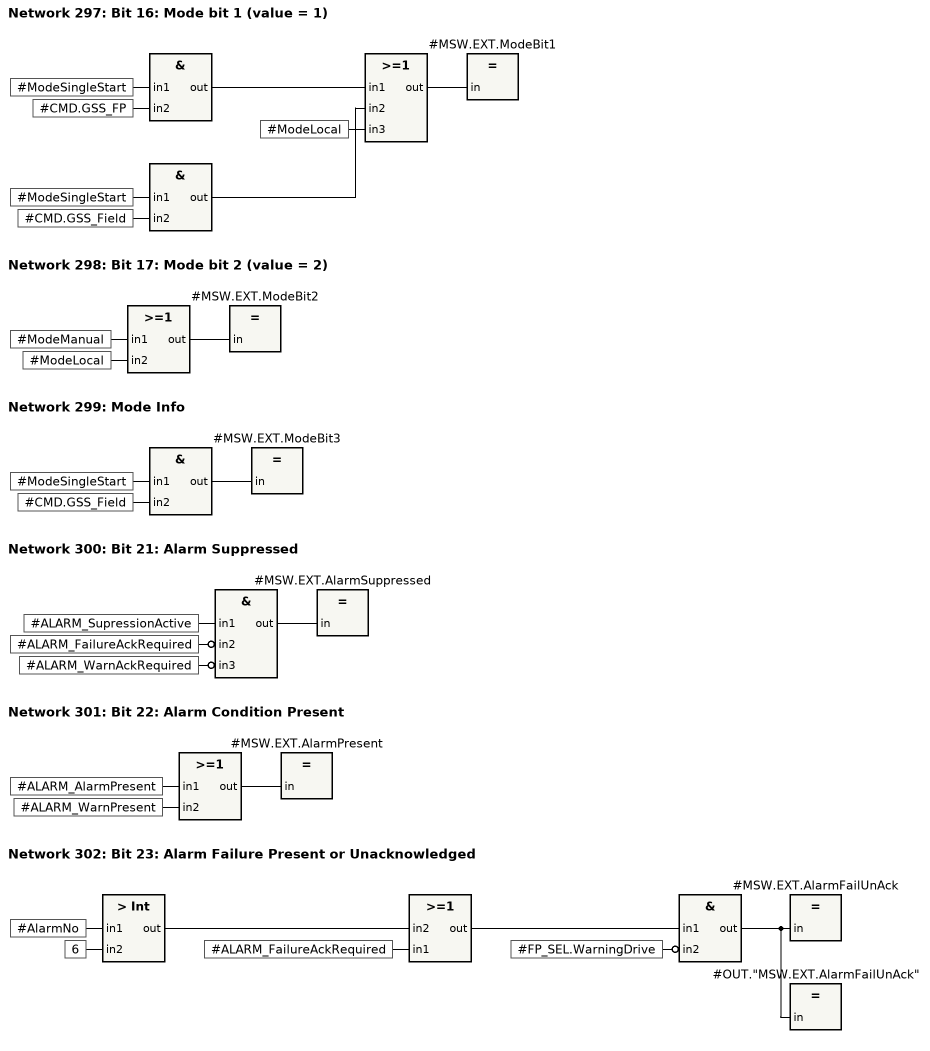
   #MSW.EXT.ModeBit1 := (#ModeSingleStart AND #CMD.GSS_FP) OR (#ModeSingleStart AND #CMD.GSS_Field) OR #ModeLocal;
END_REGION

REGION Network 298: Bit 17: Mode bit 2 (value = 2)
   #MSW.EXT.ModeBit2 := #ModeManual OR #ModeLocal;
END_REGION

REGION Network 299: Mode Info
   #MSW.EXT.ModeBit3 := #ModeSingleStart AND #CMD.GSS_Field;
END_REGION

REGION Network 300: Bit 21: Alarm Suppressed
   #MSW.EXT.AlarmSuppressed := #ALARM_SupressionActive AND NOT #ALARM_FailureAckRequired AND NOT #ALARM_WarnAckRequired;
END_REGION

REGION Network 301: Bit 22: Alarm Condition Present
   #MSW.EXT.AlarmPresent := #ALARM_AlarmPresent OR #ALARM_WarnPresent;
END_REGION

REGION Network 302: Bit 23: Alarm Failure Present or Unacknowledged
   #MSW.EXT.AlarmFailUnAck := ((#AlarmNo > 6) OR #ALARM_FailureAckRequired) AND NOT #FP_SEL.WarningDrive;
   #OUT."MSW.EXT.AlarmFailUnAck" := #MSW.EXT.AlarmFailUnAck;
END_REGION

REGION Network 303: Bit 24: Alarm Warning Present or Unacknowledged
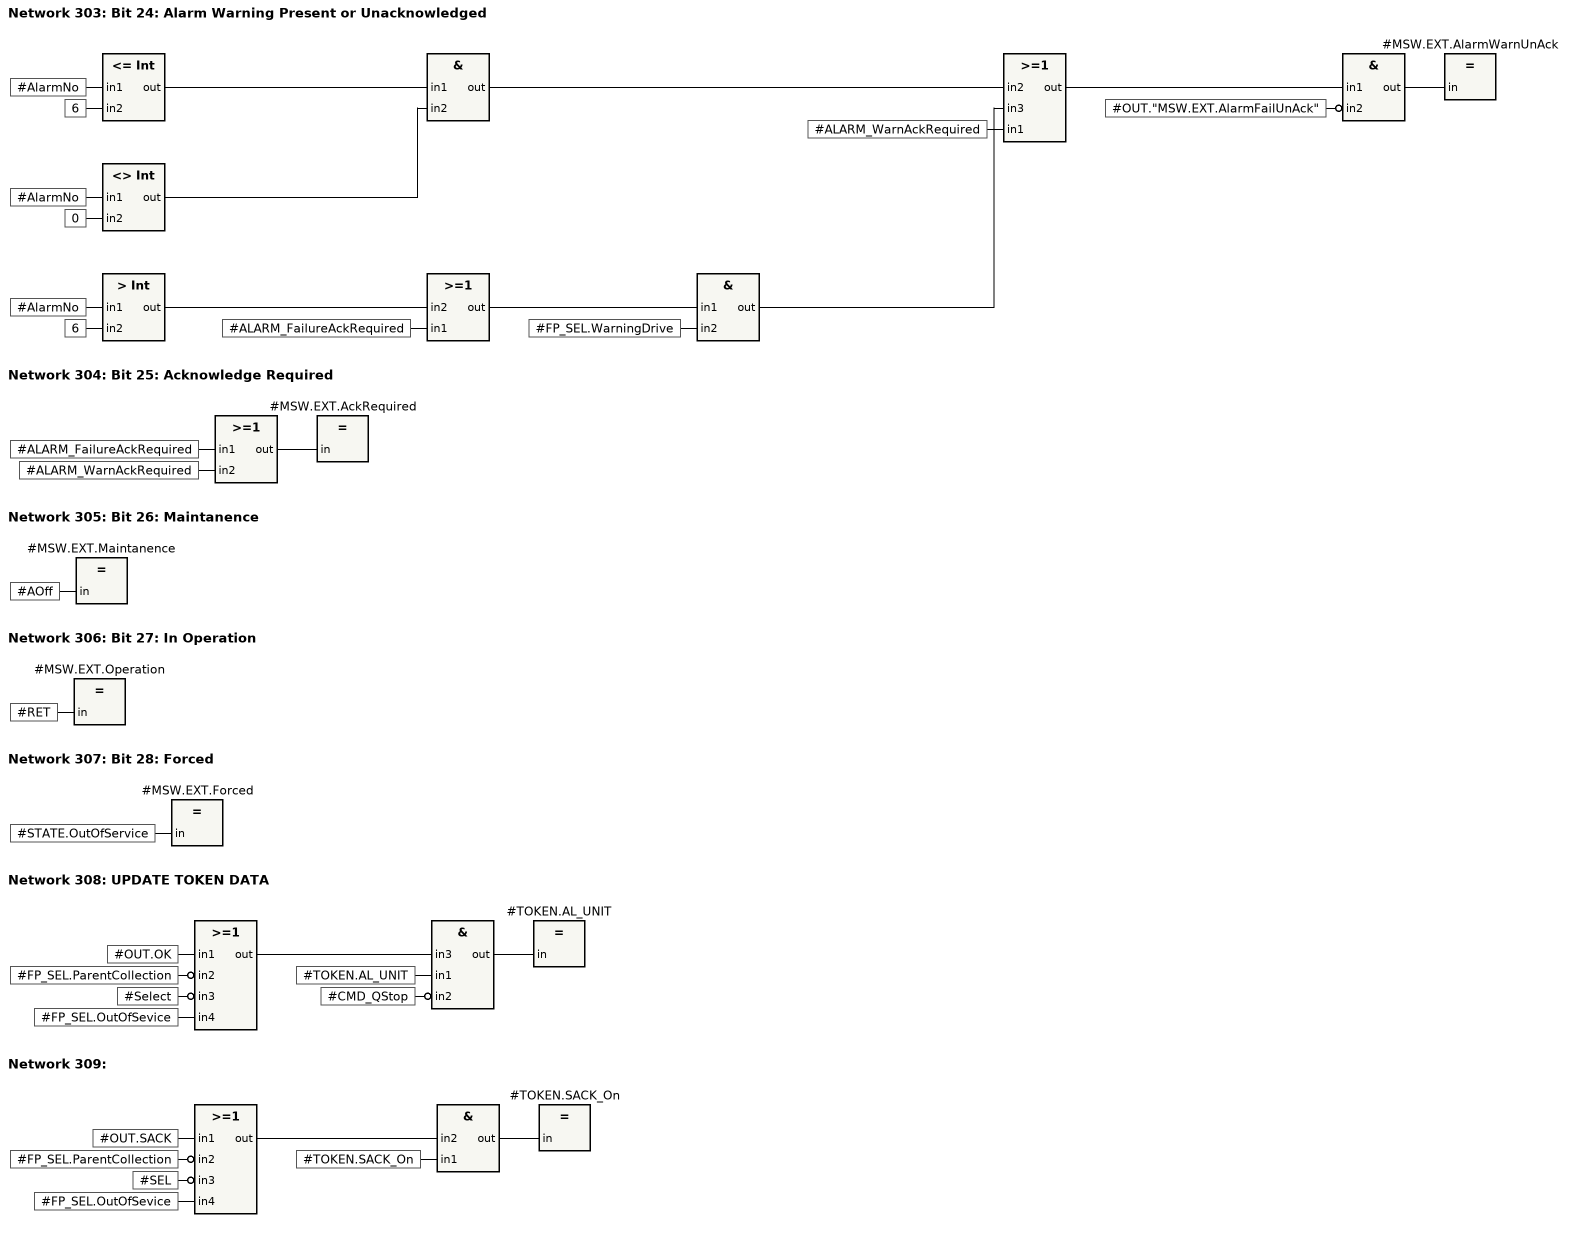
   #MSW.EXT.AlarmWarnUnAck := (((#AlarmNo <= 6) AND (#AlarmNo <> 0)) OR (((#AlarmNo > 6) OR #ALARM_FailureAckRequired) AND #FP_SEL.WarningDrive) OR #ALARM_WarnAckRequired) AND NOT #OUT."MSW.EXT.AlarmFailUnAck";
END_REGION

REGION Network 304: Bit 25: Acknowledge Required
   #MSW.EXT.AckRequired := #ALARM_FailureAckRequired OR #ALARM_WarnAckRequired;
END_REGION

REGION Network 305: Bit 26: Maintanence
   #MSW.EXT.Maintanence := #AOff;
END_REGION

REGION Network 306: Bit 27: In Operation
   #MSW.EXT.Operation := #RET;
END_REGION

REGION Network 307: Bit 28: Forced
   // Build 002 - 27 March 2018: OuOfService condition would show Force icon (bit 28)
   #MSW.EXT.Forced := #STATE.OutOfService;
END_REGION

REGION Network 308: UPDATE TOKEN DATA
   #TOKEN.AL_UNIT := (#OUT.OK OR NOT #FP_SEL.ParentCollection OR NOT #Select OR #FP_SEL.OutOfSevice) AND #TOKEN.AL_UNIT AND NOT #CMD_QStop;
END_REGION

REGION Network 309
   // Build 005 - 24.Jun.2020 (MIA-US): Replace "Select" with "SEL"
   #TOKEN.SACK_On := (#OUT.SACK OR NOT #FP_SEL.ParentCollection OR NOT #SEL OR #FP_SEL.OutOfSevice) AND #TOKEN.SACK_On;
END_REGION

REGION Network 310
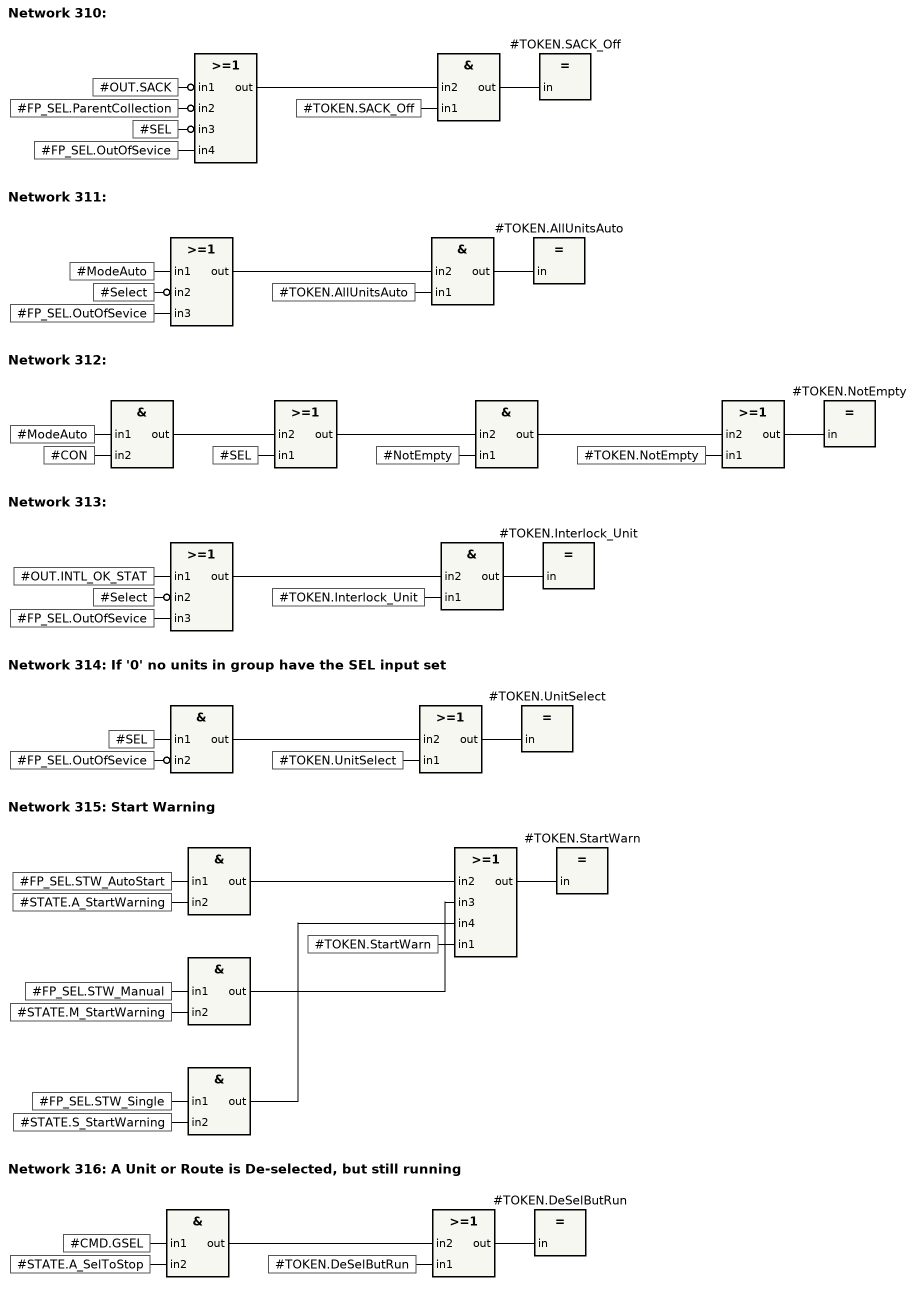
   #TOKEN.SACK_Off := (NOT #OUT.SACK OR NOT #FP_SEL.ParentCollection OR NOT #SEL OR #FP_SEL.OutOfSevice) AND #TOKEN.SACK_Off;
END_REGION

REGION Network 311
   #TOKEN.AllUnitsAuto := (#ModeAuto OR NOT #Select OR #FP_SEL.OutOfSevice) AND #TOKEN.AllUnitsAuto;
END_REGION

REGION Network 312
   #TOKEN.NotEmpty := (((#ModeAuto AND #CON) OR #SEL) AND #NotEmpty) OR #TOKEN.NotEmpty;
END_REGION

REGION Network 313
   #TOKEN.Interlock_Unit := (#OUT.INTL_OK_STAT OR NOT #Select OR #FP_SEL.OutOfSevice) AND #TOKEN.Interlock_Unit;
END_REGION

REGION Network 314: If '0' no units in group have the SEL input set
   #TOKEN.UnitSelect := (#SEL AND NOT #FP_SEL.OutOfSevice) OR #TOKEN.UnitSelect;
END_REGION

REGION Network 315: Start Warning
   #TOKEN.StartWarn := (#FP_SEL.STW_AutoStart AND #STATE.A_StartWarning) OR (#FP_SEL.STW_Manual AND #STATE.M_StartWarning) OR (#FP_SEL.STW_Single AND #STATE.S_StartWarning) OR #TOKEN.StartWarn;
END_REGION

REGION Network 316: A Unit or Route is De-selected, but still running
   #TOKEN.DeSelButRun := (#CMD.GSEL AND #STATE.A_SelToStop) OR #TOKEN.DeSelButRun;
END_REGION

REGION Network 317: Interlock
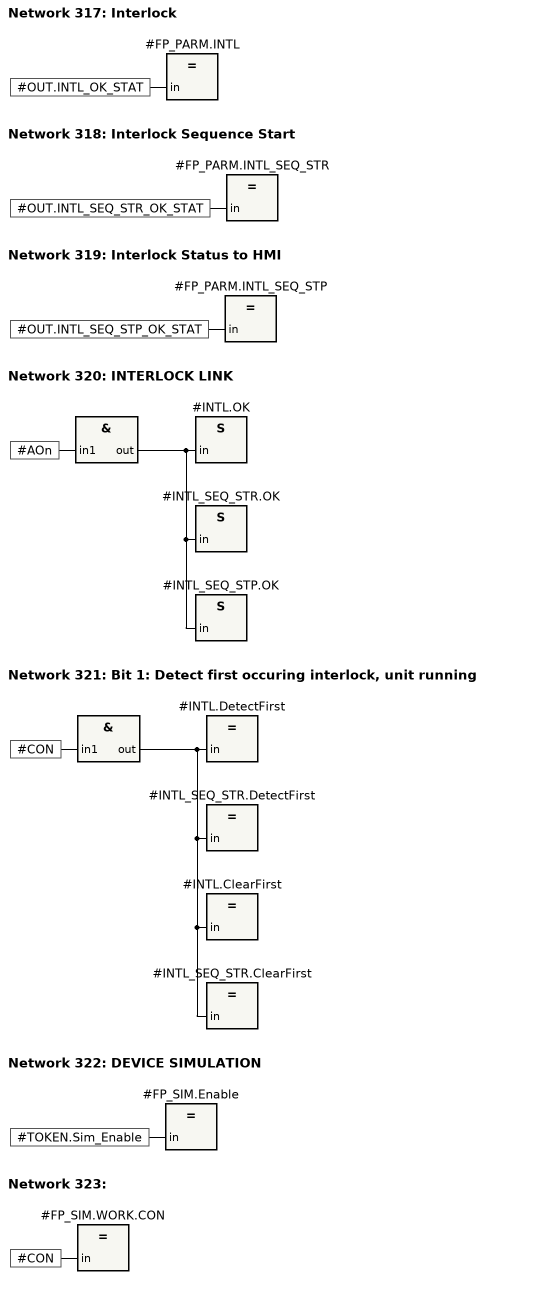
   #FP_PARM.INTL := #OUT.INTL_OK_STAT;
END_REGION

REGION Network 318: Interlock Sequence Start
   #FP_PARM.INTL_SEQ_STR := #OUT.INTL_SEQ_STR_OK_STAT;
END_REGION

REGION Network 319: Interlock Status to HMI
   #FP_PARM.INTL_SEQ_STP := #OUT.INTL_SEQ_STP_OK_STAT;
END_REGION

REGION Network 320: INTERLOCK LINK
   IF #AOn THEN
       #INTL.OK := TRUE;
       #INTL_SEQ_STR.OK := TRUE;
       #INTL_SEQ_STP.OK := TRUE;
   END_IF;
END_REGION

REGION Network 321: Bit 1: Detect first occuring interlock, unit running
   #INTL.DetectFirst := #CON;
   #INTL_SEQ_STR.DetectFirst := #CON;
   #INTL.ClearFirst := #CON;
   #INTL_SEQ_STR.ClearFirst := #CON;
END_REGION

REGION Network 322: DEVICE SIMULATION
   #FP_SIM.Enable := #TOKEN.Sim_Enable;
END_REGION

REGION Network 323
   #FP_SIM.WORK.CON := #CON;
END_REGION

REGION Network 324
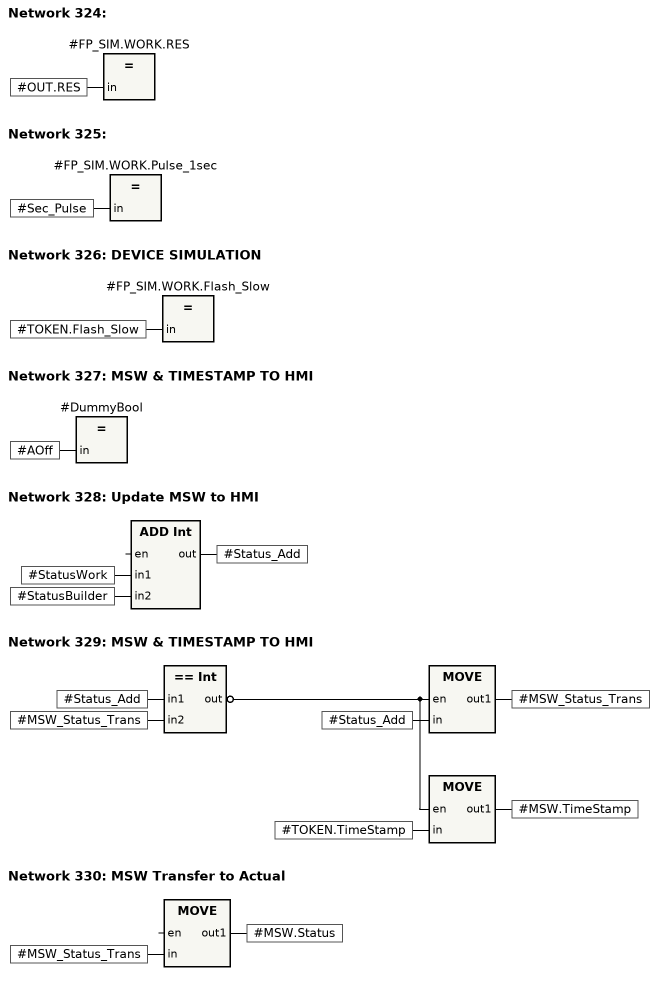
   #FP_SIM.WORK.RES := #OUT.RES;
END_REGION

REGION Network 325
   #FP_SIM.WORK.Pulse_1sec := #Sec_Pulse;
END_REGION

REGION Network 326: DEVICE SIMULATION
   #FP_SIM.WORK.Flash_Slow := #TOKEN.Flash_Slow;
END_REGION

REGION Network 327: MSW & TIMESTAMP TO HMI
   Done:
   #DummyBool := #AOff;
END_REGION

REGION Network 328: Update MSW to HMI
   #Status_Add := #StatusWork + #StatusBuilder;
END_REGION

REGION Network 329: MSW & TIMESTAMP TO HMI
   #_w1 := NOT (#Status_Add = #MSW_Status_Trans);
   IF #_w1 THEN
       #MSW_Status_Trans := #Status_Add;
       #MSW.TimeStamp := #TOKEN.TimeStamp;
   END_IF;
END_REGION

REGION Network 330: MSW Transfer to Actual
   #MSW.Status := #MSW_Status_Trans;
END_REGION

REGION Network 331: Write STAT to OUT
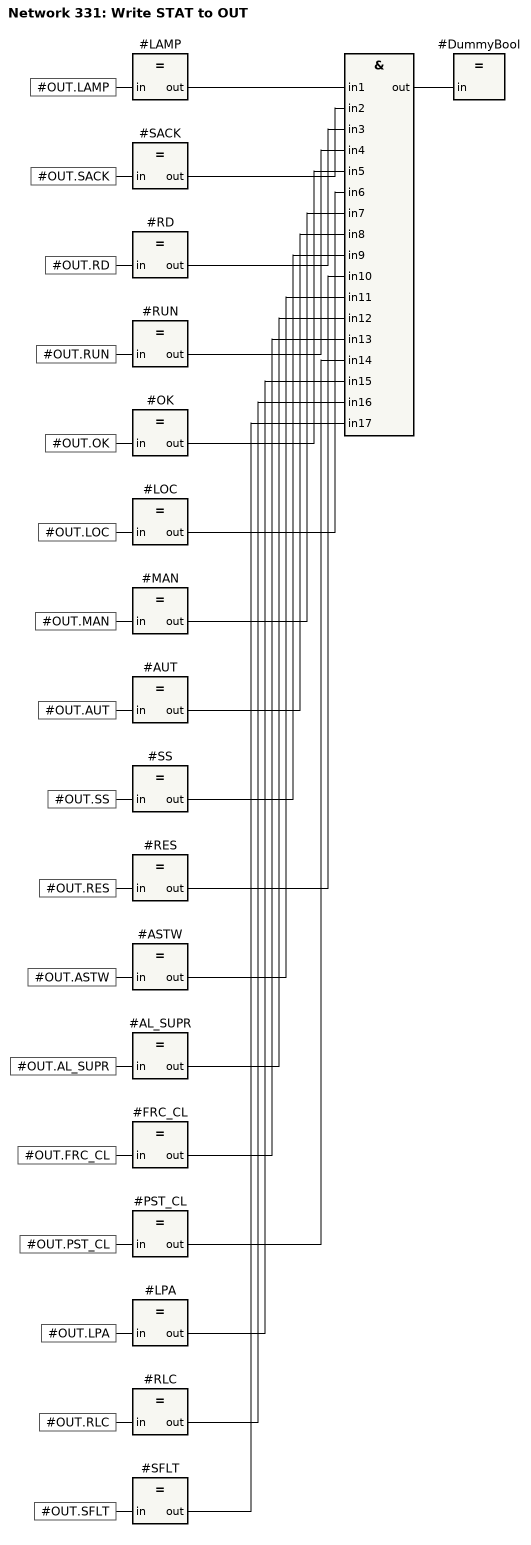
   #LAMP := #OUT.LAMP;
   #SACK := #OUT.SACK;
   #RD := #OUT.RD;
   #RUN := #OUT.RUN;
   #OK := #OUT.OK;
   #LOC := #OUT.LOC;
   #MAN := #OUT.MAN;
   #AUT := #OUT.AUT;
   #SS := #OUT.SS;
   #RES := #OUT.RES;
   #ASTW := #OUT.ASTW;
   #AL_SUPR := #OUT.AL_SUPR;
   #FRC_CL := #OUT.FRC_CL;
   #PST_CL := #OUT.PST_CL;
   #LPA := #OUT.LPA;
   #RLC := #OUT.RLC;
   #SFLT := #OUT.SFLT;
   #DummyBool := #OUT.LAMP AND #OUT.SACK AND #OUT.RD AND #OUT.RUN AND #OUT.OK AND #OUT.LOC AND #OUT.MAN AND #OUT.AUT AND #OUT.SS AND #OUT.RES AND #OUT.ASTW AND #OUT.AL_SUPR AND #OUT.FRC_CL AND #OUT.PST_CL AND #OUT.LPA AND #OUT.RLC AND #OUT.SFLT;
END_REGION
END_FUNCTION_BLOCK

FUNCTION_BLOCK "ACESYS_PFISTER_SDD"   // FB218, SCL
TITLE = ACESYS V8.0 - Build 005 - PFISTER SDD Block
{ S7_Optimized_Access := 'FALSE' }
AUTHOR : FLSmidth
FAMILY : ACESYS
NAME : PFISTER_SDD
VERSION : 8.0
   VAR_INPUT
      CMD : "ACESYS_GRP_CMD";
      SEL : Bool;
      ASTR : Bool;
      SSW : Bool;
      DOS_SP : Real;
      MEAS_SP : Real;
      OPT_VAL_RATIO : Int;
   END_VAR
   VAR_OUTPUT
      INTL : "ACESYS_INTL";
      INTL_SEQ_STR : "ACESYS_INTL";
      INTL_SEQ_STP : "ACESYS_INTL";
      LAMP : Bool;
      SACK : Bool;
      RD : Bool;
      RUN : Bool;
      OK : Bool;
      WARN : Bool;
      LOC : Bool;
      MAN : Bool;
      AUT : Bool;
      SS : Bool;
      ASTW : Bool;
      AL_SUPR : Bool;
      DOS : Bool;
      MEAS : Bool;
      FEED_Pct : Real;
      FEED_Eng : Real;
      SPEED_Pct : Real;
      SPEED_Eng : Real;
      LOAD_Pct : Real;
      TOT_Pulse : Bool;
      ERROR_CODE : Int;
      MSW : "ACESYS_HMI_STAT_32T";
   END_VAR
   VAR_IN_OUT
      TOKEN : "ACESYS_TOKEN";
   END_VAR
   VAR
      BlockInfo : Struct
         Ace_Version : Int;
         Ace_BuildNo : Int;
         State_Act : Int;
         State_Prev : Int;
         DB_Number : Int;
      END_STRUCT;
      FP_CMD : Struct
         QuickStop : Bool;
         SetUserCorr : Bool;
         Auto : Bool;
         Manual : Bool;
         Local : Bool;
         Start : Bool;
         Reset : Bool;
         AckAlarm : Bool;
         Stop : Bool;
         Measuring : Bool;
         Dosing : Bool;
         Spare_04 : Bool;
         Spare_03 : Bool;
         Spare_02 : Bool;
         Spare_01 : Bool;
         Spare_00 : Bool;
      END_STRUCT;
      FP_SEL : Struct
         STW_AutoStart : Bool;
         STW_Manual : Bool;
         STW_Single : Bool;
         STW_Local : Bool;
         ParentSupress : Bool;
         ParentCollection : Bool;
         OutOfSevice : Bool;
         Spare_00 : Bool;
         Spare_01 : Bool;
         Spare_02 : Bool;
         Spare_03 : Bool;
         Spare_04 : Bool;
         Spare_05 : Bool;
         Spare_06 : Bool;
         Spare_07 : Bool;
         Spare_08 : Bool;
      END_STRUCT;
      FP_EN : Struct
         Mode_Auto : Bool;
         Mode_Man : Bool;
         Mode_Loc : Bool;
         Mode_SS_Field : Bool;
         Mode_SS_FP : Bool;
         PB_QStop : Bool;
         Spare_00 : Bool;
         Spare_01 : Bool;
         Spare_02 : Bool;
         Spare_03 : Bool;
         Spare_04 : Bool;
         Spare_05 : Bool;
         Spare_06 : Bool;
         Spare_07 : Bool;
         Spare_08 : Bool;
         Spare_09 : Bool;
      END_STRUCT;
      FP_DIM : Struct
         Auto : Bool;
         Local : Bool;
         Manual : Bool;
         Start : Bool;
         Stop : Bool;
         QStop : Bool;
         Measuring : Bool;
         Dosing : Bool;
         Reset : Bool;
         SetUserCorr : Bool;
         Spare6 : Bool;
         Spare5 : Bool;
         Spare4 : Bool;
         Spare3 : Bool;
         Spare2 : Bool;
         Spare1 : Bool;
      END_STRUCT;
      FP_SHOW : Struct
         PB_Auto : Bool;
         PB_Local : Bool;
         PB_Manual : Bool;
         PB_Start : Bool;
         PB_Stop : Bool;
         PB_QStop : Bool;
         ACK : Bool;
         PB_Dosing : Bool;
         PB_Measuring : Bool;
         PB_Reset : Bool;
         Feedrate : Bool;
         Load : Bool;
         Speed : Bool;
         Preload : Bool;
         Current : Bool;
         Droppointload : Bool;
      END_STRUCT;
      FP_PARM : Struct
         INTL : Bool;
         INTL_SEQ_STR : Bool;
         INTL_SEQ_STP : Bool;
         CorrAccepted : Bool;
         SelectVal_Enable : Bool;
         Run : Bool;
         Spare02 : Bool;
         Spare01 : Bool;
         StartWarn_Pre : DInt;
         StartWarn_Acc : DInt;
         RunDelay_Pre : DInt;
         RunDelay_Acc : DInt;
         DelayStart_Pre : DInt;
         DelayStart_Acc : DInt;
         DelayStop_Pre : DInt;
         DelayStop_Acc : DInt;
         ReturnMon_Pre : DInt;
         ReturnMon_Acc : DInt;
         CORR_User : Real;
         Measuring_SP : Real;
         Dosing_SP : Real;
         Feedrate_SP : Real;
         Act_Feedrate : Int;
         Act_Load : Int;
         Act_Speed : Int;
         Act_Preload : Int;
         Act_Current : Int;
         Act_Droppointload : Int;
         OptValRatio : Int;
         StopReason : Int;
         PresentError : Int;
         LastError : Int;
         PresentWarning : Int;
         LastWarning : Int;
         Range_Feed : Real;
         Range_Speed : Real;
      END_STRUCT;
      FP_SIM : "ACESYS_SIM_PFISTER_SDD";
      AdapterBlock : "ACESYS_ADPT_PFISTERSDD";
      STATE : Struct
         A_AutoStart : Bool;
         A_DelayedStart : Bool;
         A_DelayedStop : Bool;
         A_Running : Bool;
         A_Selected : Bool;
         A_SelToStop : Bool;
         A_Stopping : Bool;
         A_SeqStart : Bool;
         A_SeqStop : Bool;
         A_Starting : Bool;
         A_StartWarning : Bool;
         A_Stopped : Bool;
         A_EmptyingSystem : Bool;
         S_AutoStart : Bool;
         S_Running : Bool;
         S_Starting : Bool;
         S_StartWarning : Bool;
         S_Stopped : Bool;
         S_Stopping : Bool;
         S_EmptyingSystem : Bool;
         M_Running : Bool;
         M_Starting : Bool;
         M_StartWarning : Bool;
         M_Stopped : Bool;
         M_Stopping : Bool;
         M_EmptyingSystem : Bool;
         L_Running : Bool;
         L_Stopped : Bool;
         Alarm : Bool;
         Interlock : Bool;
         EmergencyStop : Bool;
         OutOfService : Bool;
      END_STRUCT;
      ONS : Struct
         AckAlarm : Bool;
         Cmd_Auto : Bool;
         Cmd_Manual : Bool;
         Cmd_Local : Bool;
         Cmd_Start : Bool;
         Cmd_Measuring : Bool;
         Cmd_Dosing : Bool;
         GLTP : Bool;
         FP_Start_CMD : Bool;
         SetUserCorr : Bool;
         ResetTot : Bool;
         Reset : Bool;
         Sec_Pulse1 : Bool;
         Sec_Pulse2 : Bool;
      END_STRUCT;
      Pulse_Flag : Struct
         AckAlarm : Bool;
         Cmd_Auto : Bool;
         Cmd_Manual : Bool;
         Cmd_Local : Bool;
         Cmd_Start : Bool;
         Cmd_Measuring : Bool;
         Cmd_Dosing : Bool;
         GLTP : Bool;
         FP_Start_CMD : Bool;
         SetUserCorr : Bool;
         ResetTot : Bool;
         Reset : Bool;
         Sec_Pulse1 : Bool;
         Sec_Pulse2 : Bool;
      END_STRUCT;
      StatusWork : Int;
      AlarmNo : Int;
      AlarmNo_Old : Int;
      RET_VAL_Output : Int;
      RET_VAL_Input : Int;
      SelectVal_Count : Int;
      ModePointer : Int;
      DelayStart_Pre : DInt;
      DelayStart_Acc : DInt;
      DelayStop_Pre : DInt;
      DelayStop_Acc : DInt;
      StartWarn_Pre : DInt;
      StartWarn_Acc : DInt;
      RunDelay_Pre : DInt;
      RunDelay_Acc : DInt;
      ReturnMon_Pre : DInt;
      ReturnMon_Acc : DInt;
      DelayStart_Mem : DInt;
      DelayStop_Mem : DInt;
      StartWarn_Mem : DInt;
      RunDelay_Mem : DInt;
      ReturnMon_Mem : DInt;
      GWA : Bool;
      GFA : Bool;
      CMD_AckAlarm : Bool;
      CMD_Start : Bool;
      CMD_Stop : Bool;
      CMD_QStop : Bool;
      CMD_Measuring : Bool;
      CMD_Dosing : Bool;
      FromStateAuto : Bool;
      FromStateSingle : Bool;
      FromStateManual : Bool;
      FromStateLocal : Bool;
      FromStopState : Bool;
      ALARM_SupressionActive : Bool;
      ALARM_AlarmPresent : Bool;
      ALARM_WarnPresent : Bool;
      ALARM_FailureAckRequired : Bool;
      ALARM_WarnAckRequired : Bool;
      StartWarn_TT : Bool;
      StartWarn_Done : Bool;
      Rundelay_Done : Bool;
      DelayStart_Done : Bool;
      DelayStop_Done : Bool;
      ReturnMon_Done : Bool;
      Trig_RET_ALARM : Bool;
      RET_OneScan : Bool;
      NotEmpty : Bool;
      Sec_Pulse : Bool;
      Start : Bool;
      ModeAuto : Bool;
      ModeLocal : Bool;
      ModeManual : Bool;
      ModeSingleStart : Bool;
      ModeMeasuring : Bool;
      ModeDosing : Bool;
      Select : Bool;
      BitVar : Bool;
      OUT : Struct
         LAMP : Bool;
         SACK : Bool;
         RD : Bool;
         RUN : Bool;
         OK : Bool;
         WARN : Bool;
         LOC : Bool;
         MAN : Bool;
         AUT : Bool;
         SS : Bool;
         ASTW : Bool;
         AL_SUPR : Bool;
         DOS : Bool;
         MEAS : Bool;
         INTL_OK_STAT : Bool;
         INTL_SEQ_STR_OK_STAT : Bool;
         INTL_SEQ_STP_OK_STAT : Bool;
         ERROR_CODE : Int;
      END_STRUCT;
      DelayStart_Timer : TON_TIME;
      DelayStop_Timer : TON_TIME;
      StartWarn_Timer : TON_TIME;
      RunDelay_Timer : TON_TIME;
      ReturnMon_Timer : TON_TIME;
      UserCorr_Timer : TON_TIME;
      Reset_Timer : TON_TIME;
      WatchDog_Timer : TON_TIME;
   END_VAR
   VAR_TEMP
      AOn : Bool;
      AOff : Bool;
      Temp_CON : Bool;
      BusFault : Bool;
      WatchDog_Elapsed : Bool;
      WatchDog_Same : Bool;
      SelectVal_Same : Bool;
      DummyBool : Bool;
      DummyBool1 : Bool;
      DummyBool2 : Bool;
      DummyBool3 : Bool;
      DummyReal : Real;
      DummyWord : Word;
      DummyDWord : DWord;
      DummyDInt : DInt;
      DummyInt : Int;
      StatPointer_Old : Int;
      StatusBuilder : Int;
      Status_Add : Int;
      Error_Old : Int;
      Warning_Old : Int;
      AnyPtr : ANY;
      AnyStruct AT AnyPtr : Struct
         S7_ID : Byte;
         Mem_ID : Byte;
         NumberOfElements : Int;
         DB_Number : Word;
         BitPointer : DWord;
      END_STRUCT;
   END_VAR
BEGIN
   (* ----------------------------------------------------------------- Block Information -------------------------------------------------------------*)
   (* Version AND Build No *)
   #BlockInfo.Ace_Version := 80;
   #BlockInfo.Ace_BuildNo := 5;

   (* INSTANCE DB Number TO Faceplate *)
   #AnyPtr := #BitVar;
   #BlockInfo.DB_Number := WORD_TO_INT(#AnyStruct.DB_Number);

   (* Second Pulse *)
   #Pulse_Flag.Sec_Pulse1 := #TOKEN.SEC_Toggle AND NOT #ONS.Sec_Pulse1;
   #ONS.Sec_Pulse1 := #TOKEN.SEC_Toggle;

   #Pulse_Flag.Sec_Pulse2 := NOT #TOKEN.SEC_Toggle AND NOT #ONS.Sec_Pulse2;
   #ONS.Sec_Pulse2 := NOT #TOKEN.SEC_Toggle;

   #Sec_Pulse := #Pulse_Flag.Sec_Pulse1 OR #Pulse_Flag.Sec_Pulse2;
   #Pulse_Flag.ResetTot := #Sec_Pulse OR #Pulse_Flag.ResetTot;

   #OUT.INTL_OK_STAT := PEEK_BOOL(area := 16#84, dbNumber := #BlockInfo.DB_Number, byteOffset := 14, bitOffset := 0);
   #OUT.INTL_SEQ_STR_OK_STAT := PEEK_BOOL(area := 16#84, dbNumber := #BlockInfo.DB_Number, byteOffset := 16, bitOffset := 0);
   #OUT.INTL_SEQ_STP_OK_STAT := PEEK_BOOL(area := 16#84, dbNumber := #BlockInfo.DB_Number, byteOffset := 18, bitOffset := 0);

   (* ----------------------------------------------------------------- Initialization ------------------------------------------------------------- *)
   (* ---- WatchDog ---- *)

   IF #FP_SIM.Enable THEN
       #WatchDog_Same := #AdapterBlock.Togglebit_T = #FP_SIM.WORK.Togglebit;
   ELSE
       #WatchDog_Same := #AdapterBlock.Togglebit_R = #AdapterBlock.Togglebit_T;
   END_IF;

   #WatchDog_Timer(IN := NOT #WatchDog_Same,
                   PT := INT_TO_DINT(3000),
                   ET => #DummyDInt,
                   Q => #WatchDog_Elapsed);


   IF #FP_SIM.Enable THEN
       #AdapterBlock.Togglebit_T := NOT #FP_SIM.WORK.Togglebit;
   ELSE
       #AdapterBlock.Togglebit_T := NOT #AdapterBlock.Togglebit_R;
   END_IF;
   #BusFault := NOT (#FP_SIM.Enable AND  #WatchDog_Elapsed);

   (* ---- #Select ---- *)
   #Select := #CMD.GSEL AND #SEL;

   (* // ---- Init Modes ---- *)
   IF NOT #FP_EN.Mode_Auto AND NOT #FP_EN.Mode_Loc AND NOT #FP_EN.Mode_Man AND NOT #FP_EN.Mode_SS_Field AND NOT #FP_EN.Mode_SS_FP THEN
       #FP_EN.Mode_Auto := TRUE;
       #FP_EN.Mode_Man := TRUE;
       #FP_EN.Mode_Loc := TRUE;
       #FP_EN.Mode_SS_FP := TRUE;
   END_IF;

   IF NOT #CMD_Measuring AND NOT #CMD_Dosing THEN
       #CMD_Measuring := TRUE;
   END_IF;

   (* // ---- Show Push Buttons ---- *)
   #FP_SHOW.PB_Auto := NOT #FP_SEL.OutOfSevice AND #FP_EN.Mode_Auto;
   #FP_SHOW.PB_Local := NOT #FP_SEL.OutOfSevice AND #FP_EN.Mode_Loc AND #TOKEN.Loc_Enable AND NOT #TOKEN.REM_TYPE;
   #FP_SHOW.PB_Manual := NOT #FP_SEL.OutOfSevice AND #FP_EN.Mode_Man AND #TOKEN.Man_Enable;
   #FP_SHOW.PB_Start := NOT #FP_SEL.OutOfSevice AND (#FP_EN.Mode_Man OR #FP_EN.Mode_SS_FP);
   #FP_SHOW.PB_Stop := NOT #FP_SEL.OutOfSevice AND (#FP_EN.Mode_Man OR #FP_EN.Mode_SS_FP);
   #FP_SHOW.PB_QStop := NOT #FP_SEL.OutOfSevice AND #FP_EN.PB_QStop AND #TOKEN.QSTOP_FP_Unit;

   IF #FP_SIM.Enable THEN
       #FP_PARM.Run := #FP_SIM.WORK.Run;
   ELSE
       #FP_PARM.Run := #AdapterBlock.Run;
   END_IF;



   (* // ----------------------------------------------------------------- FacePlate DimOuts -------------------------------------------------------------//  *)
   (* // ---- DimOut Buttons ---- *)
   (* // Auto Button *)
   #FP_DIM.Auto := #ModeLocal OR #ModeManual;
   #FP_DIM.Auto := #FP_DIM.Auto AND NOT (#TOKEN.LOC_TYPE AND #ModeLocal AND #FP_PARM.Run);
   #FP_DIM.Auto := #FP_DIM.Auto AND NOT (#ModeLocal AND #CMD.GLTP);
   #FP_DIM.Auto := #FP_DIM.Auto AND #FP_SHOW.PB_Auto AND #TOKEN.EmergencyStop;
   (* // Manual Button *)
   #FP_DIM.Manual := #ModeLocal AND NOT #TOKEN.LOC_TYPE;
   #FP_DIM.Manual := #FP_DIM.Manual OR (#ModeLocal AND #TOKEN.LOC_TYPE AND NOT #FP_PARM.Run);
   #FP_DIM.Manual := #FP_DIM.Manual OR (#ModeAuto AND NOT #Select AND NOT #STATE.A_SelToStop AND NOT #STATE.A_Stopping AND NOT #STATE.A_Selected);
   #FP_DIM.Manual := #FP_DIM.Manual AND NOT (#ModeLocal AND #CMD.GLTP);
   #FP_DIM.Manual := #FP_DIM.Manual AND #FP_SHOW.PB_Manual AND #TOKEN.EmergencyStop;
   (* // Local Button *)
   #FP_DIM.Local := #ModeAuto AND NOT #Select AND NOT #STATE.A_SelToStop AND NOT #STATE.A_Stopping;
   #FP_DIM.Local := #FP_DIM.Local OR #ModeManual;
   #FP_DIM.Local := #FP_DIM.Local AND #FP_SHOW.PB_Local AND #TOKEN.EmergencyStop;
   (* // Stop Button *)
   CASE #ModePointer OF
       51:  // ModeAuto
           #FP_DIM.Stop := #CMD.GSEL AND NOT #SEL AND #STATE.A_SelToStop;
       52:  // ModeManual
           #FP_DIM.Stop := #OUT.INTL_SEQ_STP_OK_STAT AND #STATE.M_Running;
           #FP_DIM.Stop := #FP_DIM.Stop OR #STATE.M_StartWarning OR #STATE.M_Starting;

       53:  // ModeSingleStart 
           #FP_DIM.Stop := #STATE.S_Running OR #STATE.S_AutoStart;
           #FP_DIM.Stop := #FP_DIM.Stop AND #OUT.INTL_SEQ_STP_OK_STAT;
           #FP_DIM.Stop := #FP_DIM.Stop OR #STATE.S_StartWarning OR #STATE.S_Starting;
           #FP_DIM.Stop := #FP_DIM.Stop AND #CMD.GSS_FP;
       ELSE
           #FP_DIM.Stop := FALSE;
           ;
   END_CASE;
   // Start Button
   CASE #ModePointer OF
       52:  // ModeManual
           #FP_DIM.Start := NOT #STATE.M_Starting AND NOT #STATE.M_StartWarning AND #OUT.INTL_OK_STAT AND #OUT.INTL_SEQ_STR_OK_STAT;
       53:  // ModeSignalStart
           #FP_DIM.Start := #CMD.GSS_FP AND #FP_EN.Mode_SS_FP AND NOT #STATE.S_Starting AND NOT #STATE.S_StartWarning AND NOT #STATE.S_AutoStart AND #OUT.INTL_SEQ_STR_OK_STAT;
       ELSE
           #FP_DIM.Start := FALSE;
           ;
   END_CASE;
   #FP_DIM.Start := #FP_DIM.Start AND NOT #Start AND NOT #STATE.Alarm;
   // Quick Stop Button
   // // Build 003 - 10 MAR 2021 VIV-IN OUT.STAT variables added insread of Output //
   #FP_DIM.QStop := #FP_SHOW.PB_QStop AND (#Start OR #OUT.SACK);
   // Set User Correction Button
   #FP_DIM.SetUserCorr := NOT #FP_CMD.SetUserCorr;
   // Measuring Button
   #FP_DIM.Measuring := #TOKEN.EmergencyStop AND #ModeDosing AND NOT #Start AND NOT #STATE.Alarm;
   // Dosing Button
   #FP_DIM.Dosing := #TOKEN.EmergencyStop AND #ModeMeasuring AND NOT #Start AND NOT #STATE.Alarm;
   // Reset Button
   #FP_DIM.Reset := (#FP_PARM.PresentError <> 0 OR #FP_PARM.PresentWarning <> 0) AND NOT #FP_CMD.Reset;

   // ----------------------------------------------------------------- Operation Modes -------------------------------------------------------------// 
   // ---- Auto Mode ----
   #Pulse_Flag.Cmd_Auto := #FP_CMD.Auto AND NOT #ONS.Cmd_Auto;
   #ONS.Cmd_Auto := #FP_CMD.Auto;
   IF #Pulse_Flag.Cmd_Auto AND #FP_DIM.Auto THEN
       #ModePointer := 51;
   END_IF;
   IF #Select AND #FP_EN.Mode_Auto THEN
       #ModePointer := 51;
   END_IF;
   IF #ModePointer < 51 THEN
       #ModePointer := 51;
   END_IF;
   IF #TOKEN.FIRST_SCAN OR #FP_SEL.OutOfSevice THEN
       #ModePointer := 51;
   END_IF;
   IF NOT #ModeAuto AND NOT #ModeLocal AND NOT #ModeManual AND NOT #ModeSingleStart THEN
       #ModePointer := 51;
   END_IF;

   IF #ModeManual AND NOT #FP_SHOW.PB_Manual THEN
       #ModePointer := 51;
   END_IF;

   #Pulse_Flag.GLTP := NOT #CMD.GLTP AND NOT #ONS.GLTP;
   #ONS.GLTP := NOT #CMD.GLTP;
   IF #Pulse_Flag.GLTP AND #ModeLocal THEN
       #ModePointer := 51;
   END_IF;

   IF #ModeLocal THEN
       IF NOT #CMD.GLTP AND (NOT #FP_EN.Mode_Loc OR NOT #TOKEN.Loc_Enable) THEN
           #ModePointer := 51;
       END_IF;
   END_IF;

   IF #ModeSingleStart THEN
       IF #FP_EN.Mode_Auto THEN
           IF (NOT (#FP_EN.Mode_SS_Field AND #TOKEN.SS_Field_Enable)) AND (NOT (#FP_EN.Mode_SS_FP AND #TOKEN.SS_FP_Enable)) THEN
               #ModePointer := 51;
           END_IF;
           IF NOT #CMD.GSS_FP AND NOT #CMD.GSS_Field THEN
               #ModePointer := 51;
           END_IF;
           IF #CMD.GSS_Field AND NOT #TOKEN.SS_Field_Enable THEN
               #ModePointer := 51;
           END_IF;
           IF #CMD.GSS_FP AND NOT #TOKEN.SS_FP_Enable THEN
               #ModePointer := 51;
           END_IF;
       END_IF;
   END_IF;

   // ---- Manual Mode ----
   #Pulse_Flag.Cmd_Manual := #FP_CMD.Manual AND NOT #ONS.Cmd_Manual;
   #ONS.Cmd_Manual := #FP_CMD.Manual;
   #DummyBool := #ModeAuto AND NOT #Select AND NOT #STATE.A_SelToStop AND NOT #STATE.A_Stopping;
   #DummyBool := #DummyBool OR #ModeLocal;
   IF #Pulse_Flag.Cmd_Manual AND #FP_DIM.Manual AND #DummyBool THEN
       #ModePointer := 52;
   END_IF;
   IF #ModeAuto AND #FP_SHOW.PB_Manual AND NOT #FP_SHOW.PB_Auto THEN
       #ModePointer := 52;
   END_IF;

   //---- Single Start Mode ----
   #DummyBool1 := #ModeAuto OR #ModeLocal OR #ModeManual;
   #DummyBool1 := #DummyBool1 AND NOT #Select AND NOT #STATE.A_Stopping;
   #DummyBool1 := #DummyBool1 OR (NOT #FP_SHOW.PB_Auto AND NOT #FP_SHOW.PB_Local AND NOT #FP_SHOW.PB_Manual);
   #DummyBool2 := #FP_EN.Mode_SS_Field AND #TOKEN.SS_Field_Enable AND #CMD.GSS_Field;
   #DummyBool2 := #DummyBool2 OR (#FP_EN.Mode_SS_FP AND #TOKEN.SS_FP_Enable AND #CMD.GSS_FP);
   IF #DummyBool1 AND #DummyBool2 THEN
       #ModePointer := 53;
   END_IF;

   //---- Local Mode ----
   (* #DummyBool := #ModeAuto OR #ModeManual;
   #Pulse_Flag.Cmd_Local := #FP_CMD.Local AND NOT #ONS.Cmd_Local;
   #ONS.Cmd_Local := #FP_CMD.Local;
   #DummyBool1 := #DummyBool AND #Pulse_Flag.Cmd_Local AND #FP_DIM.Local;
   #DummyBool2 := #DummyBool AND #CMD.GLTP;
   IF NOT #STATE.A_SelToStop AND NOT #STATE.A_Stopping THEN
       IF #DummyBool1 OR #DummyBool2 AND (NOT #Select AND NOT #CMD.GSS_FP AND NOT #CMD.GSS_Field) THEN
           #ModePointer := 54;
       ELSIF #ModeAuto AND #FP_SHOW.PB_Local AND NOT #FP_SHOW.PB_Auto THEN
           #ModePointer := 54;
       END_IF;
   END_IF; *)

   IF #AdapterBlock.FieldMode OR (#FP_SIM.Enable AND #FP_SIM.WORK.FieldMode) THEN
       #ModePointer := 54;
   END_IF;

   //---- Measuring Mode ----
   #Pulse_Flag.Cmd_Measuring := #FP_CMD.Measuring AND NOT #ONS.Cmd_Measuring;
   #ONS.Cmd_Measuring := #FP_CMD.Measuring;
   IF #Pulse_Flag.Cmd_Measuring AND #FP_DIM.Measuring THEN
       #CMD_Measuring := TRUE;
       #CMD_Dosing := FALSE;
   END_IF;

   //---- Dosing Mode ----
   #Pulse_Flag.Cmd_Dosing := #FP_CMD.Dosing AND NOT #ONS.Cmd_Dosing;
   #ONS.Cmd_Dosing := #FP_CMD.Dosing;
   IF #Pulse_Flag.Cmd_Dosing AND #FP_DIM.Dosing THEN
       #CMD_Dosing := TRUE;
       #CMD_Measuring := FALSE;
   END_IF;

   //---- Modes Setting ----
   #ModeAuto := #ModePointer = 51;
   #ModeManual := #ModePointer = 52;
   #ModeSingleStart := #ModePointer = 53;
   #ModeLocal := #ModePointer = 54;

   #ModeMeasuring := #CMD_Measuring;
   #ModeDosing := #CMD_Dosing;

   #FP_CMD.Auto := #ModePointer = 51;
   #FP_CMD.Manual := #ModePointer = 52;
   #FP_CMD.Local := #ModePointer = 54;
   #FP_CMD.Measuring := #CMD_Measuring;
   #FP_CMD.Dosing := #CMD_Dosing;

   // ----------------------------------------------------------------- Faceplate Commands -------------------------------------------------------------//
   #CMD_Start := #FP_CMD.Start AND NOT #ONS.FP_Start_CMD AND #FP_DIM.Start;
   #ONS.FP_Start_CMD := #FP_CMD.Start;

   // Build 003 10 Mar 2021 - Viv-in - Inching Logic Removed //
   #CMD_Stop := #FP_CMD.Stop AND #FP_DIM.Stop;

   #CMD_QStop := #FP_CMD.QuickStop AND #FP_DIM.QStop;

   #CMD_AckAlarm := #TOKEN.Acknowledge AND NOT #ONS.AckAlarm OR #FP_CMD.AckAlarm;
   #ONS.AckAlarm := #TOKEN.Acknowledge;

   #DummyBool := #FP_CMD.SetUserCorr AND NOT #ONS.SetUserCorr;
   #ONS.SetUserCorr := #FP_CMD.SetUserCorr;

   IF #FP_DIM.SetUserCorr AND #DummyBool THEN
       #FP_CMD.SetUserCorr := TRUE;
   END_IF;

   #DummyBool := #FP_CMD.Reset AND NOT #ONS.Reset;
   #ONS.Reset := #FP_CMD.Reset;

   IF (#DummyBool OR #CMD_AckAlarm) AND #FP_DIM.Reset THEN
       #FP_CMD.Reset := TRUE;
   END_IF;

   //Reset Command
   IF #FP_CMD.Stop THEN
       #FP_CMD.Stop := FALSE;
   END_IF;

   IF #FP_CMD.QuickStop THEN
       #FP_CMD.QuickStop := FALSE;
   END_IF;

   IF #CMD_AckAlarm THEN
       #FP_CMD.AckAlarm := FALSE;
   END_IF;

   IF #CMD_AckAlarm THEN
       #FP_CMD.AckAlarm := FALSE;
   END_IF;

   // Build 003 - 10 MAR 2021 VIV-IN Inching Reset Logic removed //
   IF #FP_CMD.Start THEN
       #FP_CMD.Start := FALSE;
   END_IF;

   IF #UserCorr_Timer.Q THEN
       #FP_CMD.SetUserCorr := FALSE;
   END_IF;

   IF #FP_PARM.PresentError = 0 AND #FP_PARM.PresentWarning = 0 OR #Reset_Timer.Q THEN
       #FP_CMD.Reset := FALSE;
   END_IF;

   // ----------------------------------------------------------------- Alarm Suppression -------------------------------------------------------------//
   // // Build 003 - 10 MAR 2021 VIV-IN OUT.STAT variables added insread of Output //
   #ALARM_SupressionActive := #ModeAuto AND #FP_SEL.ParentSupress AND (#TOKEN.AlarmSuppres OR NOT #SEL);
   #AL_SUPR := #ModeAuto AND NOT #OUT.SACK AND NOT #Select;

   // ----------------------------------------------------------------- Main Logic -------------------------------------------------------------//
   // ---- Detect Mode From Last State ----
   #FromStateAuto := #BlockInfo.State_Act >= 100 AND #BlockInfo.State_Act <= 199;
   #FromStateSingle := #BlockInfo.State_Act >= 200 AND #BlockInfo.State_Act <= 299;
   #FromStateManual := #BlockInfo.State_Act >= 300 AND #BlockInfo.State_Act <= 399;
   #FromStateLocal := #BlockInfo.State_Act >= 400 AND #BlockInfo.State_Act <= 499;
   #FromStopState := #BlockInfo.State_Act >= 600 OR #BlockInfo.State_Act <= 100;
   #FromStopState := #FromStopState OR #TOKEN.FIRST_SCAN;
   #FromStopState := #FromStopState OR (#STATE.Alarm AND NOT #ALARM_AlarmPresent AND NOT #ALARM_FailureAckRequired);
   #DummyBool := #ModeAuto OR #ModeSingleStart;
   #DummyBool := #DummyBool AND NOT #Select;
   #DummyBool := #DummyBool OR #OUT.INTL_OK_STAT;
   #DummyBool := #DummyBool AND #STATE.Interlock;
   #FromStopState := #FromStopState OR #DummyBool;
   #FromStopState := #FromStopState OR (#STATE.EmergencyStop AND #TOKEN.EmergencyStop);
   #FromStopState := #FromStopState OR (#STATE.OutOfService AND NOT #FP_SEL.OutOfSevice);

   #StatPointer_Old := #BlockInfo.State_Act;

   // ---- Auto Mode ----
   IF NOT #ModeAuto THEN
       GOTO Label_SS;
   END_IF;

   // State 100: Auto - Stopped
   // // Build 003 - 10 MAR 2021 VIV-IN OUT.STAT variables added insread of Output //
   #DummyBool1 := #STATE.A_Selected OR #STATE.A_DelayedStart OR #STATE.A_Starting OR #STATE.A_StartWarning OR #STATE.A_SeqStart;
   #DummyBool1 := #DummyBool1 AND (NOT #Select OR #CMD.GSTR) AND NOT #OUT.SACK AND NOT #Select;
   #DummyBool2 := #STATE.A_Starting OR #STATE.A_StartWarning OR #STATE.A_Running;
   #DummyBool2 := #DummyBool2 AND NOT #OUT.INTL_SEQ_STR_OK_STAT;
   #DummyBool := #DummyBool1 OR #DummyBool2 OR #STATE.A_Stopping OR (#STATE.A_SeqStart AND #CMD.GSTP);
   IF #DummyBool AND NOT #FP_PARM.Run THEN
       #BlockInfo.State_Act := 100;
   ELSIF #FromStopState OR #FromStateSingle OR #FromStateManual OR #FromStateLocal OR #CMD_QStop THEN
       #BlockInfo.State_Act := 100;
   END_IF;

   // State 102: Auto - Selected
   IF (#Select AND #STATE.A_Stopped) OR (#Select AND NOT #CMD.GSTR AND #STATE.A_SeqStart) THEN
       #BlockInfo.State_Act := 102;
   END_IF;

   // State 120: Auto - Sequence Start
   IF (#Select AND #CMD.GSTR AND #STATE.A_Selected) OR (#STATE.A_DelayedStart AND NOT #OUT.INTL_SEQ_STR_OK_STAT) THEN
       #BlockInfo.State_Act := 120;
   END_IF;

   //State 104: Auto - Delayed Start
   IF #OUT.INTL_SEQ_STR_OK_STAT AND (#STATE.A_SeqStart OR (#Select AND #CMD.GSTR AND #STATE.A_Selected)) THEN
       #BlockInfo.State_Act := 104;
   END_IF;

   // State 106: Auto - Starting
   #DummyBool := #StartWarn_Done OR NOT #FP_SEL.STW_AutoStart;
   #DummyBool := #DummyBool AND #STATE.A_StartWarning;
   #DummyBool := #DummyBool OR (#STATE.A_DelayedStart AND #DelayStart_Done);
   #DummyBool := #DummyBool AND #ASTR;
   IF #DummyBool THEN
       #BlockInfo.State_Act := 106;
   END_IF;

   // State 108: Auto - Running
   #DummyBool1 := #STATE.L_Running OR #STATE.M_Running;
   #DummyBool1 := #DummyBool1 AND #Select;
   #DummyBool1 := #DummyBool1 OR #STATE.A_Starting;
   #DummyBool1 := #DummyBool1 AND #FP_PARM.Run;
   #DummyBool2 := #STATE.A_SelToStop OR #STATE.A_DelayedStop OR #STATE.A_SeqStop;
   #DummyBool2 := #DummyBool2 AND #Select;
   #DummyBool := #DummyBool1 OR #DummyBool2 OR #STATE.S_Running;
   IF #ASTR AND #DummyBool THEN
       #BlockInfo.State_Act := 108;
   END_IF;

   // State 110: Auto - Auto Start
   #DummyBool := #STATE.A_DelayedStop AND NOT #CMD_Stop;
   #DummyBool := #DummyBool OR #STATE.A_SelToStop OR #STATE.A_SeqStop OR #STATE.L_Running OR #STATE.M_Running;
   #DummyBool := #DummyBool AND #Select;
   #DummyBool := #DummyBool OR #STATE.A_DelayedStart OR #STATE.A_Starting OR #STATE.A_Running OR #STATE.A_StartWarning OR #STATE.S_AutoStart;
   IF NOT #ASTR AND #DummyBool THEN
       #BlockInfo.State_Act := 110;
   END_IF;

   // State 112: Auto - Selected to Stop
   IF NOT #Select AND (#STATE.A_Running OR #STATE.A_AutoStart OR #STATE.A_StartWarning) THEN
       #BlockInfo.State_Act := 112;
   END_IF;

   // State 122: Auto - Sequence Stop
   #DummyBool := #STATE.A_Running OR #STATE.A_AutoStart;
   #DummyBool := #DummyBool AND #Select;
   #DummyBool := #DummyBool OR #STATE.A_SelToStop OR (#STATE.A_StartWarning AND NOT #Select);
   IF #CMD.GSTP AND #DummyBool THEN
       #BlockInfo.State_Act := 122;
   ELSIF #STATE.A_DelayedStop AND NOT #OUT.INTL_SEQ_STP_OK_STAT THEN
       #BlockInfo.State_Act := 122;
   ELSIF #STATE.A_SelToStop AND #CMD.GSEL AND NOT #SEL AND #CMD_Stop THEN
       #BlockInfo.State_Act := 122;
   END_IF;

   // State 114: Auto - Delayed Stop
   IF #STATE.A_SeqStop AND #OUT.INTL_SEQ_STP_OK_STAT THEN
       #BlockInfo.State_Act := 114;
   END_IF;

   // State 116: Auto - Stopping
   IF (#STATE.A_SelToStop OR #STATE.A_DelayedStop OR #STATE.A_StartWarning) AND #CMD.GQSTP THEN
       #BlockInfo.State_Act := 116;
   ELSIF #STATE.A_DelayedStop AND #DelayStop_Done THEN
       #BlockInfo.State_Act := 116;
   ELSIF #STATE.A_StartWarning AND #CMD.GSTP AND #Select THEN
       #BlockInfo.State_Act := 116;
   ELSIF (#STATE.A_SelToStop OR #STATE.A_DelayedStop OR #STATE.A_StartWarning OR #STATE.A_Running OR #STATE.A_AutoStart OR #STATE.A_SeqStop) AND NOT #OUT.INTL_SEQ_STR_OK_STAT THEN
       #BlockInfo.State_Act := 116;
   END_IF;

   // State 118: Auto - Start Warning
   IF #ASTR AND NOT #Start AND NOT #CMD.GSTP AND (#STATE.A_AutoStart OR #STATE.A_SelToStop) THEN
       #BlockInfo.State_Act := 118;
   END_IF;

   GOTO Label_MISC;

   // ---- Single Start Mode ----
   Label_SS:
   IF NOT #ModeSingleStart THEN
       GOTO Label_MAN;
   END_IF;

   // State 200: Single Start - Stopped
   IF NOT #FP_PARM.Run AND #STATE.S_Stopping THEN
       #BlockInfo.State_Act := 200;
   ELSIF (#STATE.S_StartWarning OR #STATE.S_Starting OR #STATE.S_Running) AND NOT #OUT.INTL_SEQ_STR_OK_STAT THEN
       #BlockInfo.State_Act := 200;
   ELSIF #FromStateAuto OR #FromStateLocal OR #FromStateManual OR #FromStopState OR #CMD_QStop THEN
       #BlockInfo.State_Act := 200;
   END_IF;

   // State 202: Single Start - Start Warning
   #DummyBool := #STATE.S_AutoStart AND #ASTR AND #FP_SEL.STW_AutoStart;
   #DummyBool := #DummyBool OR (#STATE.S_Stopped AND #CMD_Start);
   IF #DummyBool AND #OUT.INTL_SEQ_STR_OK_STAT THEN
       #BlockInfo.State_Act := 202;
   END_IF;

   //State 204: Single Start - Starting
   #DummyBool := #StartWarn_Done OR NOT #FP_SEL.STW_Single;
   #DummyBool := #DummyBool AND #STATE.S_StartWarning;
   IF #DummyBool OR (#STATE.S_AutoStart AND #ASTR) THEN
       #BlockInfo.State_Act := 204;
   END_IF;

   // State 206: Single Start - Running
   IF #OUT.INTL_SEQ_STR_OK_STAT AND #FP_PARM.Run AND (#STATE.S_Starting OR #STATE.A_Running) THEN
       #BlockInfo.State_Act := 206;
   END_IF;

   // State 210: Single Start - Stopping
   #DummyBool := #STATE.S_Running OR #STATE.S_Starting OR #STATE.S_AutoStart OR #STATE.S_StartWarning;
   #DummyBool := #DummyBool AND #CMD_Stop AND #OUT.INTL_SEQ_STP_OK_STAT;
   IF #DummyBool OR #CMD_QStop THEN
       #BlockInfo.State_Act := 210;
   END_IF;

   // State 208: Single Start - Auto Start
   IF #STATE.A_AutoStart OR (NOT #ASTR AND (#STATE.S_Starting OR #STATE.S_Running)) THEN
       #BlockInfo.State_Act := 208;
   END_IF;

   GOTO Label_MISC;

   // ---- Manual Mode ----
   Label_MAN:
   IF NOT #ModeManual THEN
       GOTO Label_LOC;
   END_IF;

   // State 300: Manual - Stopped
   IF NOT #FP_PARM.Run AND #STATE.M_Stopping THEN
       #BlockInfo.State_Act := 300;
   ELSIF (#STATE.M_StartWarning OR #STATE.M_Starting OR #STATE.M_Running) AND NOT #OUT.INTL_SEQ_STR_OK_STAT THEN
       #BlockInfo.State_Act := 300;
   ELSIF #FromStopState OR #FromStateAuto OR #FromStateLocal THEN
       #BlockInfo.State_Act := 300;
   END_IF;

   // State 301: Manual - Start Warning
   IF #STATE.M_Stopped AND #CMD_Start AND #OUT.INTL_SEQ_STR_OK_STAT THEN
       #BlockInfo.State_Act := 301;
   END_IF;

   // State 303: Manual - Starting
   IF #StartWarn_Done OR NOT #FP_SEL.STW_Manual AND #STATE.M_StartWarning AND #OUT.INTL_SEQ_STR_OK_STAT THEN
       #BlockInfo.State_Act := 303;
   END_IF;

   // State 305: Manual - Running
   IF #STATE.M_Starting AND #FP_PARM.Run THEN
       #BlockInfo.State_Act := 305;
   END_IF;

   // State 307: Manual Stopping
   IF #CMD_Stop AND #OUT.INTL_SEQ_STP_OK_STAT AND #STATE.M_Running THEN
       #BlockInfo.State_Act := 307;
   ELSIF (#STATE.M_Starting OR #STATE.M_StartWarning) AND #CMD_Stop THEN
       #BlockInfo.State_Act := 307;
   ELSIF #CMD_QStop THEN
       #BlockInfo.State_Act := 307;
   END_IF;

   GOTO Label_MISC;

   // ---- Local Mode ----
   Label_LOC:
   IF NOT #ModeLocal THEN
       GOTO Label_MISC;
   END_IF;

   // State 400/405: Stopped/Running
   #DummyBool := #FromStateAuto OR #FromStateManual OR #FromStopState OR #STATE.L_Running OR #STATE.L_Stopped;
   IF #DummyBool AND NOT #FP_PARM.Run THEN
       #BlockInfo.State_Act := 400;
   END_IF;
   IF #DummyBool AND #FP_PARM.Run THEN
       #BlockInfo.State_Act := 405;
   END_IF;

   GOTO Label_MISC;

   // ---- MISC States ---
   Label_MISC:
   // State: Interlock
   #DummyBool := NOT #FP_PARM.Run OR NOT #ModeLocal;
   #DummyBool := #DummyBool AND #TOKEN.LOC_TYPE;
   #DummyBool := #DummyBool OR NOT #TOKEN.LOC_TYPE;
   // Build 003 - 10 MAR 2021 VIV-IN OUT.STAT variables added insread of Output //
   IF #DummyBool AND NOT #OUT.INTL_OK_STAT AND (#Select OR #OUT.SACK OR NOT #ModeAuto) THEN
       #BlockInfo.State_Act := 606;
   END_IF;

   // State: Alarm
   // Build 003 - 09.03.2021 (BOBO-IN): AND gate changed to OR gate //
   IF #ALARM_AlarmPresent OR #ALARM_FailureAckRequired THEN
       #BlockInfo.State_Act := 607;
   END_IF;

   // State: Out of Service
   IF #FP_SEL.OutOfSevice THEN
       #BlockInfo.State_Act := 550;
   END_IF;

   // State: Emergency Stop
   IF NOT #TOKEN.EmergencyStop THEN
       #BlockInfo.State_Act := 608;
   END_IF;

   // ---- Set State Flags ----
   #STATE.A_Stopped := #BlockInfo.State_Act = 100;
   #STATE.A_Selected := #BlockInfo.State_Act = 102;
   #STATE.A_DelayedStart := #BlockInfo.State_Act = 104;
   #STATE.A_Starting := #BlockInfo.State_Act = 106;
   #STATE.A_Running := #BlockInfo.State_Act = 108;
   #STATE.A_AutoStart := #BlockInfo.State_Act = 110;
   #STATE.A_SelToStop := #BlockInfo.State_Act = 112;
   #STATE.A_DelayedStop := #BlockInfo.State_Act = 114;
   #STATE.A_Stopping := #BlockInfo.State_Act = 116;
   #STATE.A_StartWarning := #BlockInfo.State_Act = 118;
   #STATE.A_SeqStart := #BlockInfo.State_Act = 120;
   #STATE.A_SeqStop := #BlockInfo.State_Act = 122;

   #STATE.S_Stopped := #BlockInfo.State_Act = 200;
   #STATE.S_StartWarning := #BlockInfo.State_Act = 202;
   #STATE.S_Starting := #BlockInfo.State_Act = 204;
   #STATE.S_Running := #BlockInfo.State_Act = 206;
   #STATE.S_AutoStart := #BlockInfo.State_Act = 208;
   #STATE.S_Stopping := #BlockInfo.State_Act = 210;

   #STATE.M_Stopped := #BlockInfo.State_Act = 300;
   #STATE.M_StartWarning := #BlockInfo.State_Act = 301;
   #STATE.M_Starting := #BlockInfo.State_Act = 303;
   #STATE.M_Running := #BlockInfo.State_Act = 305;
   #STATE.M_Stopping := #BlockInfo.State_Act = 307;

   #STATE.L_Stopped := #BlockInfo.State_Act = 400;
   #STATE.L_Running := #BlockInfo.State_Act = 405;

   #STATE.Interlock := #BlockInfo.State_Act = 606;
   #STATE.Alarm := #BlockInfo.State_Act = 607;
   #STATE.OutOfService := #BlockInfo.State_Act = 550;
   #STATE.EmergencyStop := #BlockInfo.State_Act = 608;

   IF #BlockInfo.State_Act <> #StatPointer_Old THEN
       #BlockInfo.State_Prev := #StatPointer_Old;
   END_IF;

   // ---- Update MSW ----
   // Build 002 - 30.09.2020 (EXTBOB): Skipped Normal MSW status update in case of Alarm Condition, Newly Added //
   IF NOT #OUT.OK THEN
       GOTO Label_MiMw;
   END_IF;

   IF #STATE.A_Stopped OR #STATE.S_Stopped OR #STATE.M_Stopped OR #STATE.L_Stopped THEN
       #StatusWork := 1;
   END_IF;

   IF #STATE.A_Selected THEN
       #StatusWork := 11;
   END_IF;

   IF #STATE.A_SeqStart THEN
       #StatusWork := 45;
   END_IF;

   IF #STATE.A_DelayedStart THEN
       #StatusWork := 51;
   END_IF;

   IF #STATE.A_Starting OR #STATE.S_Starting OR #STATE.M_Starting THEN
       #StatusWork := 91;
   END_IF;

   IF #STATE.A_Running OR #STATE.S_Running OR #STATE.M_Running OR #STATE.L_Running THEN
       #StatusWork := 81;
   END_IF;

   IF #STATE.A_AutoStart OR #STATE.S_AutoStart THEN
       #StatusWork := 61;
   END_IF;

   IF #STATE.A_SelToStop THEN
       #StatusWork := 31;
   END_IF;

   IF #STATE.A_SeqStop THEN
       #StatusWork := 66;
   END_IF;

   IF #STATE.A_DelayedStop THEN
       #StatusWork := 71;
   END_IF;

   IF #STATE.A_Stopping OR #STATE.S_Stopping OR #STATE.M_Stopping THEN
       #StatusWork := 41;
   END_IF;
   // Build 003 - 10 MAR 2021 VIV-IN OUT.STAT variables added insread of Output //
   #DummyBool := #CMD.GASTW AND #SEL AND NOT #OUT.SACK;
   IF #DummyBool OR #STATE.A_StartWarning OR #STATE.S_StartWarning OR #STATE.M_StartWarning THEN
       #StatusWork := 21;
   END_IF;

   // Build 002 - 30.09.2020 (EXTBOB): Skipped Normal MSW status update in case of Alarm Condition, Newly Added //
   Label_MiMw:

   IF #STATE.Interlock THEN
       #StatusWork := 99;
   END_IF;

   IF #STATE.OutOfService THEN
       #StatusWork := 190;
   END_IF;

   IF #STATE.EmergencyStop THEN
       #StatusWork := 200;
   END_IF;

   // ----------------------------------------------------------------- Alarm/Warning Handling -------------------------------------------------------------//
   // Read Error Code
   IF #FP_SIM.Enable THEN
       #AdapterBlock.MessageID := 0;
   END_IF;
   #OUT.ERROR_CODE := BYTE_TO_INT(#AdapterBlock.MessageID);

   IF #OUT.ERROR_CODE >= 1 AND #OUT.ERROR_CODE <= 127 THEN
       #GWA := FALSE;
   ELSE
       #GWA := TRUE;
   END_IF;

   IF #OUT.ERROR_CODE >= 128 AND #OUT.ERROR_CODE <= 255 THEN
       #GFA := FALSE;
   ELSE
       #GFA := TRUE;
   END_IF;

   // Skip Alarm
   IF NOT #TOKEN.EmergencyStop OR #FP_SEL.OutOfSevice OR #TOKEN.FIRST_SCAN THEN
       GOTO Label_Skip;
   END_IF;

   // Alarm/Warning Present
   // // Build 003 - 10 MAR 2021 VIV-IN OUT.STAT variables added insread of Output //
   #ALARM_AlarmPresent := NOT #BusFault OR NOT #SSW OR #Trig_RET_ALARM OR NOT #GFA;
   #ALARM_WarnPresent := #OUT.WARN;

   #DummyBool := NOT #ALARM_AlarmPresent AND NOT #ALARM_WarnPresent AND NOT #ALARM_FailureAckRequired AND NOT #ALARM_WarnAckRequired;
   // Skip Alarm
   IF #AlarmNo = 0 AND #DummyBool THEN
       GOTO Label_Skip;
   END_IF;
   // Clear Alarm
   IF #AlarmNo > 0 AND #DummyBool THEN
       GOTO Label_Clear;
   END_IF;
   // Acknowledge Alarm
   IF NOT #ALARM_AlarmPresent AND NOT #ALARM_WarnPresent AND (#ALARM_FailureAckRequired OR #ALARM_WarnAckRequired) THEN
       GOTO Label_Ack;
   END_IF;

   // ---- Alarm setting ----
   // Bus Fault
   IF #AlarmNo = 5 OR NOT #BusFault THEN
       #StatusWork := 201;
       #AlarmNo := 5;
       GOTO Label_Ack;
   END_IF;

   // SSW Fault
   IF #AlarmNo = 4 OR NOT #SSW THEN
       #StatusWork := 203;
       #AlarmNo := 4;
       GOTO Label_Ack;
   END_IF;
   // Return Fault
   IF #AlarmNo = 3 OR #Trig_RET_ALARM THEN
       #StatusWork := 204;
       #AlarmNo := 3;
       GOTO Label_Ack;
   END_IF;
   // GFA Fault
   IF #AlarmNo = 2 OR NOT #GFA THEN
       #StatusWork := 205;
       #AlarmNo := 2;
       GOTO Label_Ack;
   END_IF;
   //GWA Fault
   IF #AlarmNo = 1 OR NOT #GWA THEN
       #StatusWork := 206;
       #AlarmNo := 1;
       GOTO Label_Ack;
   END_IF;

   // ---- Alarm Acknowledge
   Label_Ack:
   IF #AlarmNo > #AlarmNo_Old AND NOT #ALARM_SupressionActive THEN
       IF #AlarmNo > 1 THEN
           #ALARM_FailureAckRequired := TRUE;
       ELSE
           #ALARM_WarnAckRequired := TRUE;
       END_IF;
   END_IF;

   #AlarmNo_Old := #AlarmNo;

   IF #AlarmNo = 0 OR #CMD_AckAlarm THEN
       #ALARM_FailureAckRequired := FALSE;
       #ALARM_WarnAckRequired := FALSE;
   END_IF;

   IF #AlarmNo = 0 OR #ALARM_FailureAckRequired OR #ALARM_WarnAckRequired THEN
       GOTO Label_Skip;
   END_IF;

   Label_Clear:

   CASE #AlarmNo OF
       1:
           IF #GWA THEN
               #AlarmNo := 0;
           END_IF;
       2:
           IF #GFA THEN
               #AlarmNo := 0;
           END_IF;
       3:
           IF NOT #Trig_RET_ALARM THEN
               #AlarmNo := 0;
           END_IF;
       4:
           IF #SSW THEN
               #AlarmNo := 0;
           END_IF;
       5:
           IF #BusFault THEN
               #AlarmNo := 0;
           END_IF;

   END_CASE;

   IF #ModeLocal THEN
       #ALARM_AlarmPresent := FALSE;
       #ALARM_WarnPresent := FALSE;
       #ALARM_FailureAckRequired := FALSE;
       #ALARM_WarnAckRequired := FALSE;
       #AlarmNo := 0;
   END_IF;

   IF #AlarmNo = 0 AND (NOT #ALARM_AlarmPresent AND NOT #ALARM_WarnPresent AND NOT #ALARM_FailureAckRequired AND NOT #ALARM_WarnAckRequired) THEN
       #AlarmNo_Old := 0;
   END_IF;

   Label_Skip:
   IF NOT #TOKEN.EmergencyStop OR #FP_SEL.OutOfSevice THEN
       #ALARM_FailureAckRequired := FALSE;
       #ALARM_WarnAckRequired := FALSE;
   END_IF;

   // ----------------------------------------------------------------- Timers -------------------------------------------------------------//
   // Delayed Start Timer
   "ACESYS_SecTimer_DINT"(START := #STATE.A_DelayedStart,
                          SEC := #Sec_Pulse,
                          PRE := #FP_PARM.DelayStart_Pre,
                          ACC => #FP_PARM.DelayStart_Acc,
                          DN => #DelayStart_Done,
                          TT => #DummyBool,
                          Mem := #DelayStart_Mem);

   // Delayed Stop Timer
   "ACESYS_SecTimer_DINT"(START := #STATE.A_DelayedStop,
                          SEC := #Sec_Pulse,
                          PRE := #FP_PARM.DelayStop_Pre,
                          ACC => #FP_PARM.DelayStop_Acc,
                          DN => #DelayStop_Done,
                          TT => #DummyBool,
                          Mem := #DelayStop_Mem);

   // Start Warning Timer
   "ACESYS_SecTimer_DINT"(START := #STATE.A_StartWarning OR #STATE.S_StartWarning OR #STATE.M_StartWarning,
                          SEC := #Sec_Pulse,
                          PRE := #FP_PARM.StartWarn_Pre,
                          ACC => #FP_PARM.#StartWarn_Acc,
                          DN => #StartWarn_Done,
                          TT => #DummyBool,
                          Mem := #StartWarn_Mem);

   // Run Delay Timer
   "ACESYS_SecTimer_DINT"(START := #Start AND #FP_PARM.Run,
                          SEC := #Sec_Pulse,
                          PRE := #FP_PARM.#RunDelay_Pre,
                          ACC => #FP_PARM.#RunDelay_Acc,
                          DN => #Rundelay_Done,
                          TT => #DummyBool,
                          Mem := #RunDelay_Mem);

   // Return Monitoring Fault
   "ACESYS_SecTimer_DINT"(START := (#Start AND NOT #FP_PARM.Run) OR (NOT #Start AND #FP_PARM.Run),
                          SEC := #Sec_Pulse,
                          PRE := #FP_PARM.ReturnMon_Pre,
                          ACC => #FP_PARM.ReturnMon_Acc,
                          DN => #ReturnMon_Done,
                          TT => #DummyBool,
                          Mem := #ReturnMon_Mem);

   // Return Monitoring alarm not consider in Local Mode
   #Trig_RET_ALARM := #Start AND NOT #FP_PARM.Run AND #RET_OneScan;
   #Trig_RET_ALARM := #Trig_RET_ALARM OR #ReturnMon_Done;
   #Trig_RET_ALARM := #Trig_RET_ALARM AND NOT #ModeLocal;

   #RET_OneScan := #FP_PARM.Run;

   // Set User Correction Timer
   #UserCorr_Timer(IN := #FP_CMD.SetUserCorr,
                   PT := INT_TO_DINT(1000));

   // Reset Timer
   #Reset_Timer(IN := #FP_CMD.Reset,
                PT := INT_TO_DINT(2000));

   // ----------------------------------------------------------------- Stop Reasons -------------------------------------------------------------//

   #Temp_CON := #STATE.A_SelToStop OR #STATE.A_DelayedStop OR #STATE.A_SeqStop;
   #Temp_CON := #Temp_CON AND #ASTR;
   #Temp_CON := #Temp_CON OR #STATE.A_Starting OR #STATE.A_Running OR #STATE.S_Starting OR #STATE.S_Running OR #STATE.M_Starting OR #STATE.M_Running;
   #Temp_CON := #Temp_CON OR (#STATE.L_Running AND NOT #TOKEN.LOC_TYPE);

   IF #Temp_CON AND #Start THEN
       #FP_PARM.StopReason := 0;
       GOTO Label_S_R;
   END_IF;

   IF #FP_PARM.StopReason <> 0 AND NOT #Temp_CON AND NOT #Start THEN
       GOTO Label_S_R;
   END_IF;

   // Unknown Reason
   #FP_PARM.StopReason := 99;

   // Emergency Stop
   IF #TOKEN.EmergencyStop THEN
       #FP_PARM.StopReason := 12;
   END_IF;

   // Unit Alarm
   IF #ALARM_AlarmPresent THEN
       #FP_PARM.StopReason := 11;
   END_IF;

   // Interlock
   IF #OUT.INTL_OK_STAT THEN
       #FP_PARM.StopReason := 10;
   END_IF;

   // Sequence Interlock
   IF #Start AND NOT #OUT.INTL_SEQ_STR_OK_STAT THEN
       #FP_PARM.StopReason := 9;
   END_IF;

   // Quick Stop 
   IF #CMD_QStop AND #Start THEN
       #FP_PARM.StopReason := 6;
   END_IF;

   //Change to Auto Mode
   IF #ModeAuto AND (#FromStateLocal OR #FromStateManual) THEN
       #FP_PARM.StopReason := 5;
   END_IF;

   // Faceplate Stop 
   IF #CMD_Stop AND #Start AND (#ModeManual OR #ModeSingleStart AND #CMD.GSS_FP OR #CMD_QStop AND #TOKEN.QSTOP_FP_Unit) THEN
       #FP_PARM.StopReason := 3;
   END_IF;

   // Normal Stop
   IF #CMD.GSTP AND #STATE.A_Stopping THEN
       #FP_PARM.StopReason := 1;
   END_IF;

   Label_S_R:
   #Start := #Temp_CON;
   #AdapterBlock.CmdStart := #Temp_CON;

   // ---- Write/Read Bus Data ----
   // Write
   #AdapterBlock.CmdDosingMode := #CMD_Dosing;
   #AdapterBlock.CmdMeasuringMode := #CMD_Measuring;
   #AdapterBlock.CmdAcknowledge := #FP_CMD.Reset;
   //#AdapterBlock.CmdStart := #CMD_Start;
   #AdapterBlock.CmdCorrection := #FP_CMD.SetUserCorr;
   #AdapterBlock.DosingSetpoint := REAL_TO_INT(#DOS_SP * 100);
   #AdapterBlock.SpeedSetpoint := REAL_TO_INT(#MEAS_SP * 100);
   #AdapterBlock.RemoteCorrection := REAL_TO_INT(#FP_PARM.CORR_User * 100);
   // Read
   IF #FP_SIM.Enable THEN
       #MEAS := #FP_SIM.WORK.MeasuringMode;
       #DOS := #FP_SIM.WORK.DosingMode;
       #FP_PARM.CorrAccepted := #FP_SIM.WORK.CorrectionDone;
   ELSE
       #MEAS := #AdapterBlock.MeasuringMode;
       #DOS := #AdapterBlock.DosingMode;
       #FP_PARM.CorrAccepted := #AdapterBlock.CorrectionDone;
   END_IF;



   // Analog Input 
   #FP_PARM.Measuring_SP := #MEAS_SP;
   #FP_PARM.Dosing_SP := #DOS_SP;
   #FP_PARM.OptValRatio := #OPT_VAL_RATIO;
   #FP_PARM.Feedrate_SP := #FP_PARM.Dosing_SP * #FP_PARM.Range_Feed;
   //Optional value read
   #FP_PARM.SelectVal_Enable := #FP_SHOW.Preload OR #FP_SHOW.Current OR #FP_SHOW.Droppointload;
   #SelectVal_Same := #AdapterBlock.SelectVals = #AdapterBlock.CmdSelectVals;

   IF #WatchDog_Same THEN

       IF #FP_PARM.SelectVal_Enable THEN

           IF #AdapterBlock.CmdSelectVals = 0 AND #AdapterBlock.SelectVals = 0 THEN
               IF #SelectVal_Count < #FP_PARM.OptValRatio THEN
                   #FP_PARM.Act_Feedrate := #AdapterBlock.Feedrate * (REAL_TO_INT(#FP_PARM.Range_Feed / 100));
                   #FP_PARM.Act_Speed := #AdapterBlock.Speed / 10;
                   #FP_PARM.Act_Load := #AdapterBlock.Load / 100;
                   #SelectVal_Count := #SelectVal_Count + 1;
               ELSE
                   #AdapterBlock.CmdSelectVals := TRUE;
                   #SelectVal_Count := 0;
               END_IF;
           END_IF;

           IF #AdapterBlock.CmdSelectVals = 1 AND #AdapterBlock.SelectVals = 1 THEN
               #FP_PARM.Act_Preload := #AdapterBlock.Preload / 100;
               #FP_PARM.Act_Current := #AdapterBlock.Current / 10;
               #FP_PARM.Act_Droppointload := #AdapterBlock.Droppointload / 100;
               #AdapterBlock.CmdSelectVals := FALSE;
           END_IF;

       ELSE
           #AdapterBlock.CmdSelectVals := FALSE;
           #FP_PARM.Act_Feedrate := #AdapterBlock.Feedrate * (REAL_TO_INT(#FP_PARM.Range_Feed / 100));
           #FP_PARM.Act_Speed := #AdapterBlock.Speed / 10;
           #FP_PARM.Act_Load := #AdapterBlock.Load / 100;
       END_IF;

   END_IF;




   // ----------------------------------------------------------------- Output -------------------------------------------------------------//
   // Build 003 - 10 MAR 2021 VIV-IN OUT.STAT variables added insread of Output //
   #SACK := #OUT.SACK;
   #WARN := #OUT.WARN;
   #LAMP := #OUT.LAMP;
   #OK := #OUT.OK;
   #RUN := #OUT.RUN;
   #RD := #OUT.RD;
   #AUT := #ModeAuto;
   #LOC := #ModeLocal;
   #MAN := #ModeManual;
   #SS := #ModeSingleStart;
   #MEAS := #ModeMeasuring;
   #DOS := #ModeDosing;
   #WARN := NOT #GWA;
   #ASTW := #OUT.ASTW;
   #TOT_Pulse := #AdapterBlock.ToltalizerPulse;

   // Analog Output
   #FEED_Pct := INT_TO_REAL(#AdapterBlock.Feedrate / 100);
   #FEED_Eng := INT_TO_REAL(#AdapterBlock.Feedrate / 100) * #FP_PARM.Range_Feed;
   #SPEED_Pct := INT_TO_REAL(#AdapterBlock.Speed / 10) / #FP_PARM.Range_Speed;
   #SPEED_Eng := INT_TO_REAL(#AdapterBlock.Speed / 10);
   #LOAD_Pct := INT_TO_REAL(#AdapterBlock.Load / 100);

   // Error/Warning
   // Save Error/Warning from last scan
   #Error_Old := #FP_PARM.PresentError;
   #Warning_Old := #FP_PARM.PresentWarning;

   // OUT.Struct Move //
   // // Build 003 - 10 MAR 2021 VIV-IN OUT.STAT variables added insread of Output //
   #OUT.LAMP := (#ALARM_FailureAckRequired AND #TOKEN.Flash_Fast) OR (NOT #ALARM_FailureAckRequired AND #TOKEN.Flash_Slow);
   #OUT.LAMP := #OUT.LAMP AND #STATE.Alarm OR #FP_PARM.Run;
   #OUT.SACK := #STATE.A_Starting OR #STATE.A_Running OR #STATE.A_AutoStart OR #STATE.A_StartWarning OR #STATE.A_SelToStop OR #STATE.A_DelayedStop OR #STATE.A_SeqStop OR #STATE.A_Stopping;
   #OUT.SACK := #OUT.SACK OR #STATE.S_Starting OR #STATE.S_Running OR #STATE.S_StartWarning;
   #OUT.SACK := #OUT.SACK OR #STATE.M_Starting OR #STATE.M_Running OR #STATE.M_StartWarning;
   #OUT.SACK := #OUT.SACK OR #STATE.L_Running;
   #OUT.OK := NOT #ALARM_AlarmPresent AND NOT #ALARM_FailureAckRequired;
   #OUT.RUN := #Start AND #FP_PARM.Run;
   #OUT.RD := #Rundelay_Done AND (#ModeAuto OR #ModeLocal OR #ModeManual OR #ModeSingleStart);
   #OUT.ASTW := #STATE.A_StartWarning OR #STATE.S_StartWarning OR #STATE.M_StartWarning;
   #OUT.ASTW := #SEL AND #CMD.GASTW OR #OUT.ASTW AND NOT #StartWarn_Done;
   #ERROR_CODE := #OUT.ERROR_CODE;


   IF NOT #GWA THEN
       #FP_PARM.PresentWarning := #OUT.ERROR_CODE;
   END_IF;
   IF NOT #GFA THEN
       #FP_PARM.PresentError := #OUT.ERROR_CODE;
   END_IF;

   IF #OUT.ERROR_CODE = 0 THEN
       #FP_PARM.PresentError := 0;
       #FP_PARM.PresentWarning := 0;
   END_IF;

   IF #FP_PARM.PresentWarning <> #Warning_Old THEN
       #FP_PARM.LastWarning := #Warning_Old;
   END_IF;

   IF #FP_PARM.PresentError <> #Error_Old THEN
       #FP_PARM.LastError := #Error_Old;
   END_IF;

   // Update Boolean Data in MSW
   IF #OUT.SACK AND NOT #ASTR AND NOT #FP_PARM.Run THEN
       #StatusBuilder := WORD_TO_INT(16#8000);
   ELSE
       #StatusBuilder := 0;
   END_IF;

   IF #FP_PARM.Run THEN
       #StatusBuilder := 4096;
   ELSIF #ModeAuto OR #ModeSingleStart THEN
       #StatusBuilder := 4096;
   END_IF;

   #StatusBuilder := #StatusBuilder;

   // Mode Info
   #MSW.EXT.ModeBit1 := #ModeSingleStart AND #CMD.GSS_FP OR #ModeSingleStart AND #CMD.GSS_Field OR #ModeLocal; // Bit 16
   #MSW.EXT.ModeBit2 := #ModeManual OR #ModeLocal; // Bit 17
   #MSW.EXT.ModeBit3 := #ModeSingleStart AND #CMD.GSS_Field; // Bit 18

   // Define alarm bits
   #MSW.EXT.AlarmSuppressed := #ALARM_SupressionActive AND NOT #ALARM_FailureAckRequired AND NOT #ALARM_WarnAckRequired; // Bit 21: Alarm Suppressed
   #MSW.EXT.AlarmPresent := #ALARM_AlarmPresent OR #ALARM_WarnPresent; // Bit 22: Alarm present
   #MSW.EXT.AlarmFailUnAck := #AlarmNo > 1 OR #ALARM_FailureAckRequired; // Bit 23: Alarm Failure Present or Unacknowledged
   // Build 003 - 10 MAR 2021 VIV-IN Warning Acknowldge required logic corrected //
   #DummyBool := #AlarmNo = 1 OR #ALARM_WarnAckRequired;
   #MSW.EXT.AlarmWarnUnAck := #DummyBool AND #MSW.EXT.AlarmFailUnAck; // Bit24: Alarm Warn Present/Unack
   #MSW.EXT.AckRequired := #ALARM_FailureAckRequired OR #ALARM_WarnAckRequired; //Bit 25: Acknowledge Required

   // Define mode bits
   #MSW.EXT.Maintanence := FALSE; // Bit 26: Maintenence
   #MSW.EXT.Operation := #FP_PARM.Run; // Bit 27: Operation
   #MSW.EXT.Forced := #STATE.OutOfService; // Bit 28: Forced

   // Update MSW to HMI
   #Status_Add := #StatusBuilder + #StatusWork;
   IF #Status_Add <> #MSW.Status THEN
       #MSW.Status := #Status_Add;
       #MSW.TimeStamp := #TOKEN.TimeStamp;
   END_IF;

   // Update Token Data
   // // Build 003 - 10 MAR 2021 VIV-IN OUT.STAT variables added insread of Output //
   // // Build 004 - 06 May 2021 BOBO-IN Token.Al_Unit AND logic corrected //
   #TOKEN.AL_UNIT := (#OUT.OK OR NOT #FP_SEL.ParentCollection OR NOT #Select OR #FP_SEL.OutOfSevice) AND #TOKEN.AL_UNIT AND NOT #CMD_QStop;

   // // Build 004 - 06 May 2021 BOBO-IN Token.Sack_On AND logic corrected //
   #TOKEN.SACK_On := #TOKEN.SACK_On AND (#OUT.SACK OR NOT #FP_SEL.ParentCollection OR NOT #Select OR #FP_SEL.OutOfSevice);

   // // Build 003 - 10 MAR 2021 VIV-IN OUT.STAT variables added insread of Output //
   // // Build 004 - 06 May 2021 BOBO-IN Token.Sack_Off AND logic corrected //
   #TOKEN.SACK_Off := #TOKEN.SACK_Off AND (NOT #OUT.SACK OR NOT #FP_SEL.ParentCollection OR NOT #SEL OR #FP_SEL.OutOfSevice);

   #TOKEN.AllUnitsAuto := #TOKEN.AllUnitsAuto AND (#ModeAuto OR NOT #Select OR #FP_SEL.OutOfSevice);
   #TOKEN.NotEmpty := #TOKEN.NotEmpty OR #NotEmpty AND (#SEL OR #ModeAuto AND #Start);
   #TOKEN.Interlock_Unit := #TOKEN.Interlock_Unit AND (#OUT.INTL_OK_STAT OR NOT #Select OR #FP_SEL.OutOfSevice);
   #TOKEN.UnitSelect := #TOKEN.UnitSelect OR #SEL AND NOT #FP_SEL.OutOfSevice;
   #TOKEN.DeSelButRun := #TOKEN.DeSelButRun OR #CMD.GSEL AND #STATE.A_SelToStop;

   #DummyBool1 := #FP_SEL.STW_AutoStart AND #STATE.A_StartWarning;
   #DummyBool2 := #FP_SEL.STW_Manual AND #STATE.M_StartWarning;
   #DummyBool3 := #FP_SEL.STW_Single AND #STATE.S_StartWarning;
   #TOKEN.StartWarn := #TOKEN.StartWarn OR #DummyBool1 OR #DummyBool2 OR #DummyBool3;

   // Interlock Status to HMI
   #FP_PARM.INTL := #OUT.INTL_OK_STAT;
   #FP_PARM.INTL_SEQ_STR := #OUT.INTL_SEQ_STR_OK_STAT;
   #FP_PARM.INTL_SEQ_STP := #OUT.INTL_SEQ_STP_OK_STAT;

   // Interlock Link
   #INTL.OK := TRUE;
   #INTL_SEQ_STR.OK := TRUE;
   #INTL_SEQ_STP.OK := TRUE;

   #INTL.DetectFirst := #Start;
   #INTL.ClearFirst := #Start;
   #INTL_SEQ_STR.DetectFirst := #Start;
   #INTL_SEQ_STR.ClearFirst := #Start;

   // Device Simulation
   #FP_SIM.Enable := #TOKEN.Sim_Enable;
   #FP_SIM.DosingMode := #CMD_Dosing;
   #FP_SIM.MeasuringMode := #CMD_Measuring;
   #FP_SIM.Start := #Start;
   #FP_SIM.CorrectionDone := #FP_CMD.SetUserCorr;
   #FP_SIM.ToggleBit := #AdapterBlock.Togglebit_T;
END_FUNCTION_BLOCK

FUNCTION_BLOCK "ACESYS_PID"   // FB220, FBD
TITLE = ACESYS V8.0 - Build 003 - PID Controller
{ S7_Optimized_Access := 'FALSE' }
AUTHOR : FLSmidth
FAMILY : ACESYS
NAME : PID
VERSION : 8.0
   VAR_INPUT
      PV : Real;   // Process Value (0-100%)
      PV_OK : Bool;   // Process Value ok
      INV : Bool;   // Invert operation
      AUTO_HLC : Bool;   // HLC Mode: "0" = Manual "1" = Auto
      AUTO_FR : Bool;   // Force to Auto Mode
      MAN_FR : Bool;   // Force to Manual Mode
      CAS_FR : Bool;   // Force to Cascade Setpoint
      INT_FR : Bool;   // Force to Internal Setpoint
      FR1_FR : Bool;   // Force 1 Request
      FR2_FR : Bool;   // Force 2 Request
      FR3_FR : Bool;   // Force 3 Request
      CAS_SP : Real;   // Cascade Setpoint
      FR1_SP : Real;   // Force 1 Setpoint
      FR2_SP : Real;   // Force 2 Setpoint
      FR3_SP : Real;   // Force 3 Setpoint
      FF : Real;   // Feed Forward (0-100%)
      CYCLE : Int;   // Cycle Time
   END_VAR
   VAR_OUTPUT
      CV : Real;   // PID Output (0-100%)
      AINORM : Real;   // PV Normalized 0-100%
      SPNORM : Real;   // SP Normalized 0-100%
      AUTO : Bool;   // Controller in Auto Mode
      MAN : Bool;   // Controller in Manual Mode
      CASC : Bool;   // Controller in Cascade (auto) Mode
      MSW : "ACESYS_HMI_STAT_32T";   // Status to HMI
   END_VAR
   VAR_IN_OUT
      SPA : Real;   // Auto Setpoint
      SPM : Real;   // Manual Sepoint
      SPA_HLC : Real;   // Auto Setpoint High-Level-Control
      SPM_HLC : Real;   // Manual Sepoint High-Level-Control
      TOKEN : "ACESYS_TOKEN";
      HLC_LINK : "ACESYS_HLC_LINK";
   END_VAR
   VAR
      BlockInfo : Struct
         Ace_Version : Int;   // Acesys Block Version Number
         Ace_BuildNo : Int;   // Acesys Block Build Number
         State_Act : Int;   // Actual State Number
         State_Prev : Int;   // Previous State Number
         DB_Number : Int;   // Block Instance DB Number
      END_STRUCT;
      FP_CMD : Struct   // Faceplate Commands
         AutoTune_Start : Bool;
         AutoTune_Cancel : Bool;
         AutoTune_Abort : Bool;
         AutoTune_Accept : Bool;
         AutoTune_Steady : Bool;
         AutoTune_Start_SUT : Bool;
         AutoTune_Start_TIR : Bool;
         AckAlarm : Bool;
         Manual : Bool;
         Auto : Bool;
         Internal : Bool;
         Cascade : Bool;
         LastSPA : Bool;
         AutoTune_Undo : Bool;
         AutoTune_Ack : Bool;
         Spare_07 : Bool;
      END_STRUCT;
      FP_SEL : Struct
         HLC_GRP01 : Bool;   // Member of HLC Group 1
         HLC_GRP02 : Bool;   // Member of HLC Group 2
         HLC_GRP03 : Bool;   // Member of HLC Group 3
         HLC_GRP04 : Bool;   // Member of HLC Group 4
         HLC_GRP05 : Bool;   // Member of HLC Group 5
         HLC_GRP06 : Bool;   // Member of HLC Group 6
         HLC_GRP07 : Bool;   // Member of HLC Group 7
         HLC_GRP08 : Bool;   // Member of HLC Group 8
         HLC_GRP09 : Bool;   // Member of HLC Group 9
         HLC_GRP10 : Bool;   // Member of HLC Group 10
         PARA_SET1 : Bool := TRUE;   // PID Parametre set 1
         PARA_SET2 : Bool;   // PID Parametre set 2
         PARA_SET3 : Bool;   // PID Parametre set 3
         PARA_SET4 : Bool;   // PID Parametre set 4
         Spare2 : Bool;
         Spare1 : Bool;
      END_STRUCT;
      FP_EN : Struct   // Faceplate Commands
         Mode_Auto : Bool := TRUE;
         Mode_Cascade : Bool;
         DevFault : Bool;
         Spare_11 : Bool;
         HLC_Track : Bool;
         PV_Track : Bool;
         Spare_10 : Bool;
         Spare_09 : Bool;
         Spare_08 : Bool;
         Spare_07 : Bool;
         Spare_06 : Bool;
         Spare_05 : Bool;
         Spare_04 : Bool;
         Spare_03 : Bool;
         Spare_02 : Bool;
         Spare_01 : Bool;
      END_STRUCT;
      FP_DIM : Struct   // Faceplate Commands
         Manual : Bool;
         Auto : Bool;
         Internal : Bool;
         Cascade : Bool;
         LastSP : Bool;
         AutoTune_Start : Bool;
         AutoTune_Cancel : Bool;
         AutoTune_Accept : Bool;
         AutoTune_Abort : Bool;
         AutoTune_Start_TIR : Bool;
         AutoTune_Ack : Bool;
         AutoTune_Undo : Bool;
         AutoTune_Start_SUT : Bool;
         Spare_03 : Bool;
         Spare_02 : Bool;
         Spare_01 : Bool;
      END_STRUCT;
      FP_SHOW : Struct   // Faceplate Commands
         PB_Manual : Bool;
         PB_Auto : Bool;
         PB_Internal : Bool;
         PB_Cascade : Bool;
         PB_LastSP : Bool;
         Spare_11 : Bool;
         Spare_10 : Bool;
         Spare_09 : Bool;
         Spare_08 : Bool;
         Spare_07 : Bool;
         Spare_06 : Bool;
         Spare_05 : Bool;
         Spare_04 : Bool;
         Spare_03 : Bool;
         Spare_02 : Bool;
         Spare_01 : Bool;
      END_STRUCT;
      FP_PARM : Struct
         IN_Min : Real;   // Min Range for Input (SPA + PV)
         IN_Max : Real := 100.0;   // Max Range for Input (SPA + PV)
         OUT_Min_Lim : Real;   // Min Output Limit (0-100%)
         OUT_Max_Lim : Real := 100.0;   // Max Output Limit (0-100%)
         OUT_Min_HMI : Real;   // Min Range for Output (HMI Display)
         OUT_Max_HMI : Real := 100.0;   // Max Range for Output (HMI Display)
         GAIN_1 : Real := 0.5;   // Proportional gain 1
         GAIN_2 : Real := 0.5;   // Proportional gain 2
         GAIN_3 : Real := 0.5;   // Proportional gain 3
         GAIN_4 : Real := 0.5;   // Proportional gain 4
         TI_1 : Real := 30.0;   // Reset time 1
         TI_2 : Real := 30.0;   // Reset time 2
         TI_3 : Real := 30.0;   // Reset time 3
         TI_4 : Real := 30.0;   // Reset time 4
         TD_1 : Real;   // Derivative time 1
         TD_2 : Real;   // Derivative time 2
         TD_3 : Real;   // Derivative time 3
         TD_4 : Real;   // Derivative time 4
         FF_Factor : Real := 100.0;   // Feed Forward Factor (0-100%)
         FF_Actual : Real;
         LastSPA : Real;   // Last AUto Setpoint
         DeadBand_High : Real := 0.1;   // Deadband Upper Limit
         DeadBand_Low : Real := -0.1;   // Deadband Low Limit
         DevFault_Limit : Real := 5.0;   // Deviation Fault Limit (%)
         DevFault_Time_PRE : Int := 30;   // Deviation Fault Delay Time (sec) PRE
         DevFault_Time_ACC : Int := 30;   // Deviation Fault Delay Time (sec) ACC
         AutoTune_Length : Real := 300.0;   // Max Tune Time Length
         AutoTune_MinStep : Real := 10.0;   // Min Setpoint Step
         AutoTune_MaxCV : Real := 10.0;   // Auto Tune Output Calculated
         AutoTune_P : Real;   // Auto Tune: P
         AutoTune_I : Real;   // Auto Tune: I
         AutoTune_D : Real;   // Auto Tune: D
         AutoTune_WaitStep : Bool;
         AutoTune_Running : Bool;
         AutoTune_AcceptToAuto : Bool;
         AutoTune_TimeOut : Bool;
         AutoTune_IncreaseCV : Bool;
         AutoTune_OK : Bool;
         AutoTune_DecreaceCV : Bool;
         AutoTUne_NotOk : Bool;
         AutoTUne_DnotRequired : Bool;
         AutoTune_PIDorPI : Bool;
         Spare_06 : Bool;
         Spare_05 : Bool;
         Spare_04 : Bool;
         Spare_03 : Bool;
         Spare_02 : Bool;
         Spare_01 : Bool;
      END_STRUCT;
      FP_PARM_TIA : Struct
         AutoTune_Progress : Real;   // Progress of Tuning in %
         AutoTune_CancelTuningLevel : Real := 10.0;   // Permissible delta from original SP
         AutoTune_SUT_Phase : Int;   // Current Phase of PreTuning
         AutoTune_TIR_Phase : Int;   // Current Phase of FineTuning
         AutoTune_TIA_FP : Int;   // =100: TIA Faceplate / <>100: S7 Faceplate
         AutoTune_SUT_TuneRule_0 : Bool := true;   // PID Chien, Hrones, Reswick
         AutoTune_SUT_TuneRule_1 : Bool;   // PI Chien, Hrones, Reswick
         AutoTune_SUT_Running : Bool;   // PreTuning Running
         AutoTune_TIR_TuneRule_0 : Bool := true;   // PID Automatic
         AutoTune_TIR_TuneRule_1 : Bool;   // PID Fast
         AutoTune_TIR_TuneRule_2 : Bool;   // PID Slow
         AutoTune_TIR_TuneRule_3 : Bool;   // PID Ziegler-Nichols
         AutoTune_TIR_TuneRule_4 : Bool;   // PI Ziegler-Nichols
         AutoTune_TIR_TuneRule_5 : Bool;   // P Ziegler-Nichols
         AutoTune_TIR_Running : Bool;   // FineTuning Running
         ErrorBit00 : Bool;   // PV Out of Range
         ErrorBit02 : Bool;   // Process Oscillation not Maintained
         ErrorBit03 : Bool;   // PV Too Close to SP
         ErrorBit04 : Bool;   // SP Changed During Tuning
         ErrorBit05 : Bool;   // PreTuning not Allowed While FineTuning
         ErrorBit07 : Bool;   // PV unexpected behavior
         ErrorBit08 : Bool;   // FineTuning Invalid Calculation
         ErrorBit09 : Bool;   // Invalid Process Value
         ErrorBit10 : Bool;   // Output Calculation Failed
         ErrorBit11 : Bool;   // Sampling Time Error
         ErrorBit12 : Bool;   // Invalid Setpoint
         ErrorBit16 : Bool;   // Invalid Manual Value
         ErrorBit17 : Bool;   // Invalid Substitute Output
         ErrorBit18 : Bool;   // Invalid Disturbance
         WarningBit00 : Bool;   // Inflection Point not Found
         WarningBit02 : Bool;   // SP Limited
         WarningBit03 : Bool;   // System Properties Missing
         WarningBit04 : Bool;   // PID Mode Could not be Changed
         WarningBit05 : Bool;   // Sampling Limited by OB Call
         WarningBit06 : Bool;   // PV Out of Warning Limits
         WarningBit07 : Bool;   // Invalid Mode
         WarningBit08 : Bool;   // Manual Value Limited
         WarningBit09 : Bool;   // Tuning Rule not Supported
         WarningBit12 : Bool;   // Substitute Output Out of Range
         SpareBool14 : Bool;
         SpareBool13 : Bool;
         SpareBool12 : Bool;
         SpareBool11 : Bool;
         SpareBool10 : Bool;
         SpareBool09 : Bool;
         SpareBool08 : Bool;
         SpareBool07 : Bool;
         SpareBool06 : Bool;
         SpareBool05 : Bool;
         SpareBool04 : Bool;
         SpareBool03 : Bool;
         SpareBool02 : Bool;
         SpareBool01 : Bool;
      END_STRUCT;
      STATE : Struct
         AUTO_Int : Bool;
         AUTO_Casc : Bool;
         AUTO_HLC : Bool;
         MAN : Bool;
         MAN_HLC : Bool;
         FR1 : Bool;
         FR2 : Bool;
         FR3 : Bool;
      END_STRUCT;
      ONS : Struct
         FP_Auto1 : Bool;
         FP_Auto2 : Bool;
         FP_Man : Bool;
         FP_Int : Bool;
         FP_Casc : Bool;
         PARA_SET1 : Bool := TRUE;   // PID Parametre set 1
         PARA_SET2 : Bool;   // PID Parametre set 2
         PARA_SET3 : Bool;   // PID Parametre set 3
         PARA_SET4 : Bool;   // PID Parametre set 4
         LastSPA1 : Bool;
         LastSPA2 : Bool;
         SecPulse1 : Bool;
         SecPulse2 : Bool;
         AckAlarm : Bool;
         AutoTuneStart1 : Bool;
         AutoTuneStart2 : Bool;
         AutoTuneAdaptOn : Bool;
         AutoTuneAccept : Bool;
         AutoTuneAcceptAuto : Bool;
         AutoTuneAccepted : Bool;
         PID_ModeChange : Bool;
         Self_Auto : Bool;
         Self_Man : Bool;
         SpareBool03 : Bool;
         TunePhase4 : Bool;
         SUT_TuneRule_0 : Bool;
         SUT_TuneRule_1 : Bool;
         TIR_TuneRule_0 : Bool;
         TIR_TuneRule_1 : Bool;
         TIR_TuneRule_2 : Bool;
         TIR_TuneRule_3 : Bool;
         TIR_TuneRule_4 : Bool;
         TIR_TuneRule_5 : Bool;
         AutoTune_Undo : Bool;
      END_STRUCT;
      LastSPSelected : Bool;
      ALARM_AlarmPresent : Bool;
      ALARM_FailureAckRequired : Bool;
      DevFault_Time_Done : Bool;
      CMD_AckAlarm : Bool;
      AutoTuneAdaptOn : Bool;
      AutoTuneMAN_ON : Bool;
      AutoTuneQMan : Bool;   // Auto Tune
      AutoTuneForceToAuto : Bool;
      AutoTuneSavePar : Bool;   // Auto Tune Save Parameters
      SR_AutoTuneAdaptOn : Bool;
      OutDB_High : Bool;
      OutDB_Low : Bool;
      AutoTune_Toggle : Bool;
      From_Pid_ErrorBits : DWord;
      DevFault_Time_Men : Int;
      StatusWork : Int;
      AlarmNo : Int;
      AlarmNo_Old : Int;
      DI_PID : PID_Compact;
      MSW_Status : Int;
   END_VAR
   VAR_TEMP
      AOn : Bool;   // Always On
      AOff : Bool;   // Always Off
      HLC_Selected : Bool;   // HLC Control Active
      DummyBool : Bool;
      Sec_Pulse : Bool;
      StatPointer_Old : Int;
      DummyReal : Real;
      SPA_Norm : Real;
      SPM_Norm : Real;
      PV_Norm : Real;
      P_Real : Real;
      I_Real : Real;
      D_Real : Real;
      To_PID_P : Real;
      To_PID_I : Real;
      TO_PID_D : Real;
      Error_Norm : Real;   // Calculated Error Normalized
      From_Pid_CV : Real;
      DummyDint : DInt;
      ErrorBits_Array : Array[0..31] of Bool;
      WarningBits_Array : Array[0..31] of Bool;
   END_VAR
   VAR_TEMP   // added for the SCL form of the ladder/FBD networks
      _w1 : Bool;
      _w2 : Bool;
      _w3 : Bool;
      _w4 : Bool;
      _w5 : Bool;
      _w6 : Bool;
      _w7 : Bool;
      _w8 : Bool;
   END_VAR
BEGIN

REGION Network 1: Always On/Off
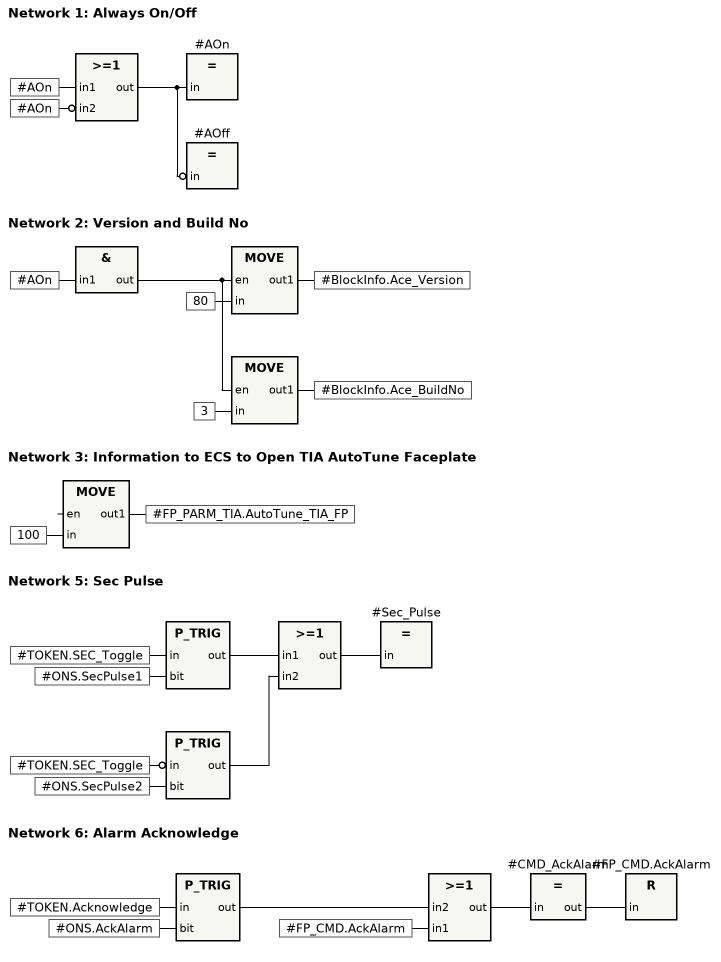
   #AOn := #AOn OR NOT #AOn;
   #AOff := NOT #AOn;
END_REGION

REGION Network 2: Version and Build No
   IF #AOn THEN
       #BlockInfo.Ace_Version := 80;
       #BlockInfo.Ace_BuildNo := 3;
   END_IF;
END_REGION

REGION Network 3: Information to ECS to Open TIA AutoTune Faceplate
   // Offset 234 corresponds to AlarmNo in S7 PID DB
   #FP_PARM_TIA.AutoTune_TIA_FP := 100;
END_REGION

REGION Network 4 (STL): Instance DB Number to Faceplate
         L     DINO;
         T     #BlockInfo.DB_Number;
END_REGION

REGION Network 5: Sec Pulse
   #_w1 := #TOKEN.SEC_Toggle AND NOT #ONS.SecPulse1;   // rising edge
   #ONS.SecPulse1 := #TOKEN.SEC_Toggle;
   #_w2 := NOT #TOKEN.SEC_Toggle AND NOT #ONS.SecPulse2;   // rising edge
   #ONS.SecPulse2 := NOT #TOKEN.SEC_Toggle;
   #Sec_Pulse := #_w1 OR #_w2;
END_REGION

REGION Network 6: Alarm Acknowledge
   #_w1 := #TOKEN.Acknowledge AND NOT #ONS.AckAlarm;   // rising edge
   #ONS.AckAlarm := #TOKEN.Acknowledge;
   #CMD_AckAlarm := #_w1 OR #FP_CMD.AckAlarm;
   IF #CMD_AckAlarm THEN #FP_CMD.AckAlarm := FALSE; END_IF;
END_REGION

REGION Network 7: HLC Control Active
   // >>>>> HLC ACTIVE <<<<<
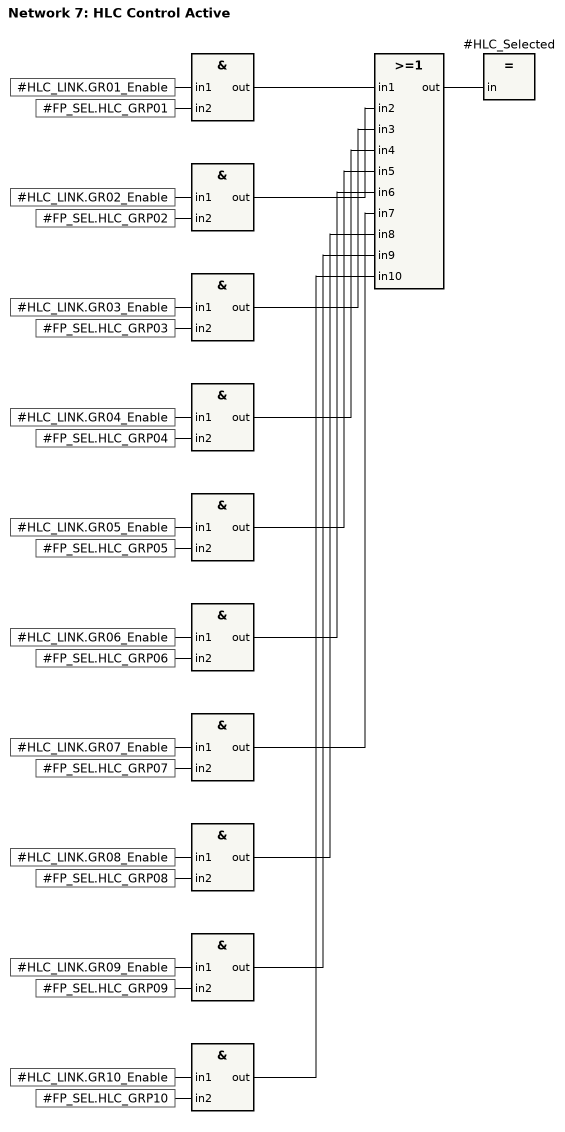
   #HLC_Selected := (#HLC_LINK.GR01_Enable AND #FP_SEL.HLC_GRP01) OR (#HLC_LINK.GR02_Enable AND #FP_SEL.HLC_GRP02) OR (#HLC_LINK.GR03_Enable AND #FP_SEL.HLC_GRP03) OR (#HLC_LINK.GR04_Enable AND #FP_SEL.HLC_GRP04) OR (#HLC_LINK.GR05_Enable AND #FP_SEL.HLC_GRP05) OR (#HLC_LINK.GR06_Enable AND #FP_SEL.HLC_GRP06) OR (#HLC_LINK.GR07_Enable AND #FP_SEL.HLC_GRP07) OR (#HLC_LINK.GR08_Enable AND #FP_SEL.HLC_GRP08) OR (#HLC_LINK.GR09_Enable AND #FP_SEL.HLC_GRP09) OR (#HLC_LINK.GR10_Enable AND #FP_SEL.HLC_GRP10);
END_REGION

REGION Network 8: Show Faceplate Pushbuttons
   // >>>>> SHOW PUSH BUTTONS ON FACEPLATE <<<<<
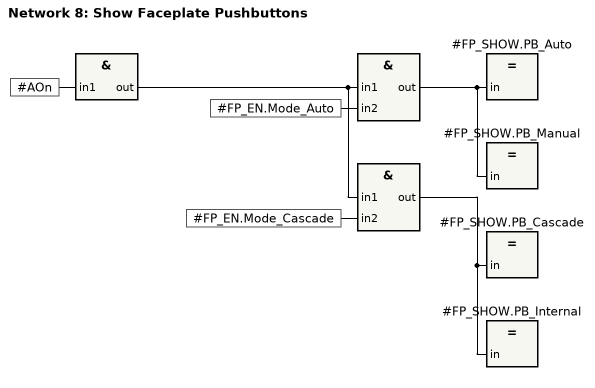
   #FP_SHOW.PB_Auto := #AOn AND #FP_EN.Mode_Auto;
   #FP_SHOW.PB_Manual := #FP_SHOW.PB_Auto;
   #FP_SHOW.PB_Cascade := #AOn AND #FP_EN.Mode_Cascade;
   #FP_SHOW.PB_Internal := #FP_SHOW.PB_Cascade;
END_REGION

REGION Network 9: Dim Out Faceplate Pushbuttons
   // >>>>> DIMOUT BUTTONS ON FACEPLATE <<<<<
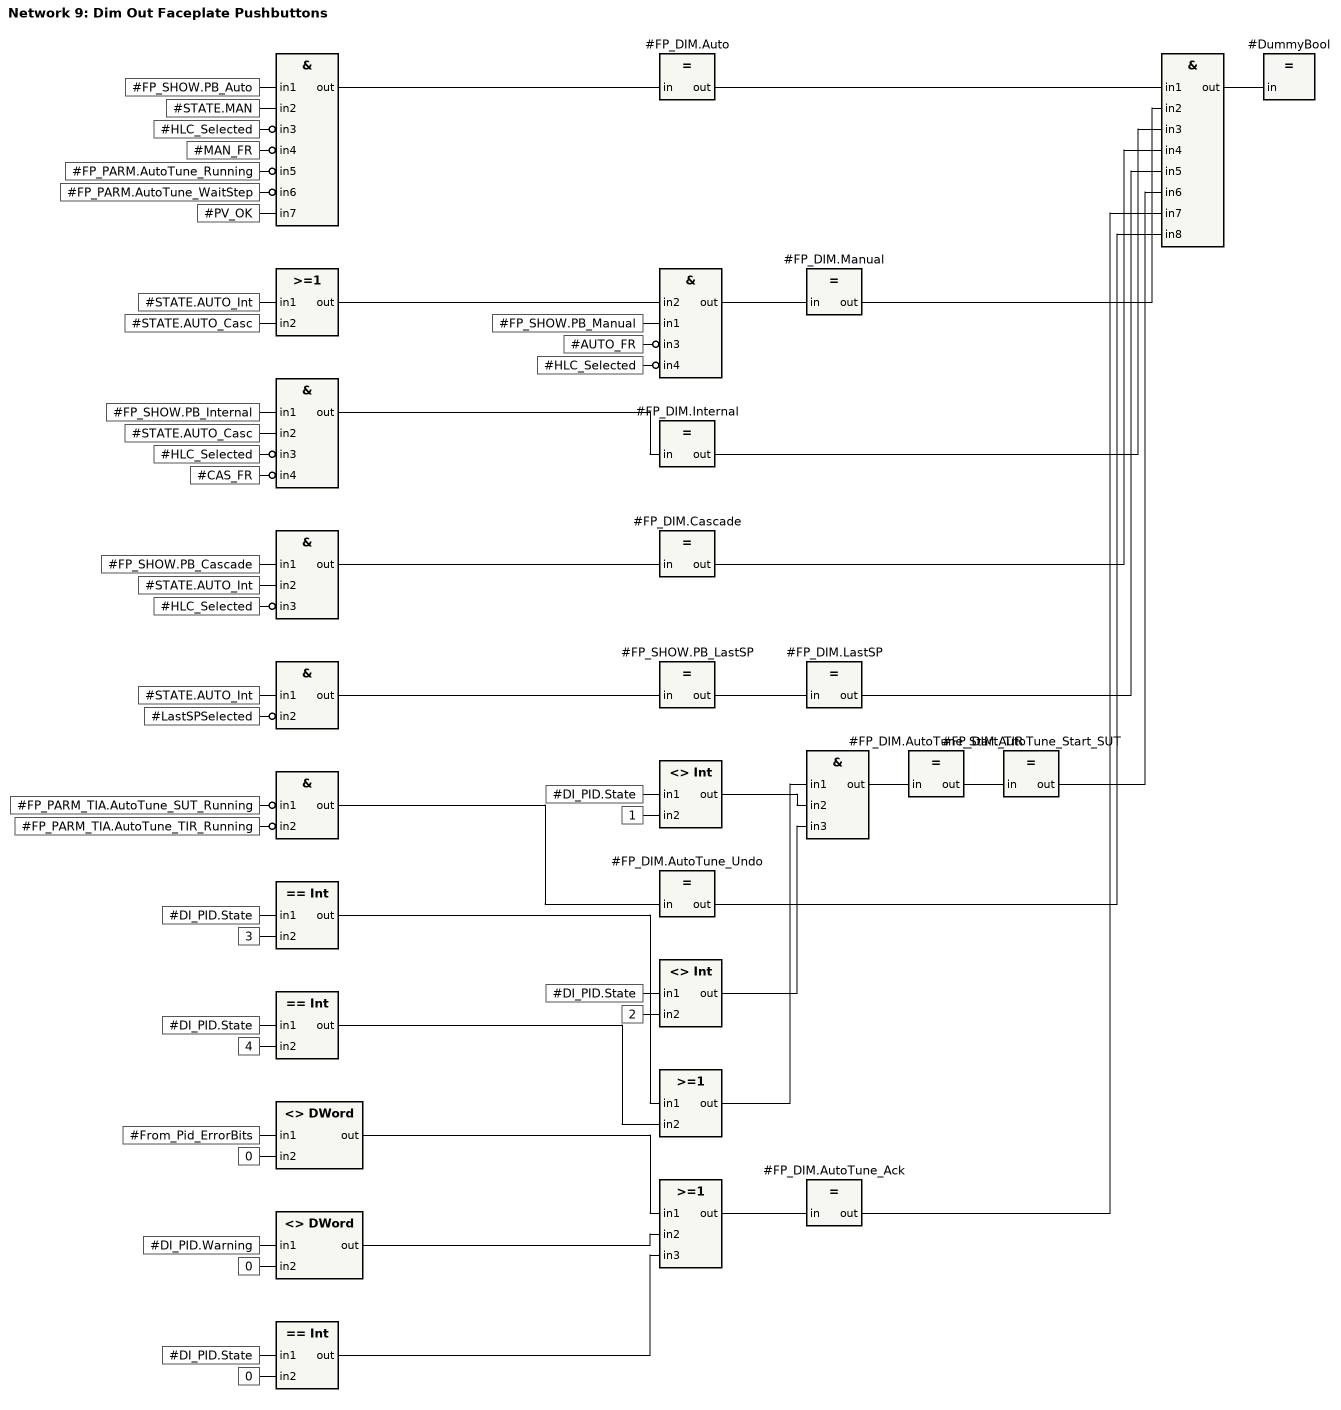
   #FP_DIM.Auto := #FP_SHOW.PB_Auto AND #STATE.MAN AND NOT #HLC_Selected AND NOT #MAN_FR AND NOT #FP_PARM.AutoTune_Running AND NOT #FP_PARM.AutoTune_WaitStep AND #PV_OK;
   #FP_DIM.Manual := (#STATE.AUTO_Int OR #STATE.AUTO_Casc) AND #FP_SHOW.PB_Manual AND NOT #AUTO_FR AND NOT #HLC_Selected;
   #FP_DIM.Internal := #FP_SHOW.PB_Internal AND #STATE.AUTO_Casc AND NOT #HLC_Selected AND NOT #CAS_FR;
   #FP_DIM.Cascade := #FP_SHOW.PB_Cascade AND #STATE.AUTO_Int AND NOT #HLC_Selected;
   #FP_SHOW.PB_LastSP := #STATE.AUTO_Int AND NOT #LastSPSelected;
   #FP_DIM.LastSP := #FP_SHOW.PB_LastSP;
   #FP_DIM.AutoTune_Start_TIR := ((#DI_PID.State = 3) OR (#DI_PID.State = 4)) AND (#DI_PID.State <> 1) AND (#DI_PID.State <> 2);
   #FP_DIM.AutoTune_Start_SUT := #FP_DIM.AutoTune_Start_TIR;
   #FP_DIM.AutoTune_Ack := (#From_Pid_ErrorBits <> 0) OR (#DI_PID.Warning <> 0) OR (#DI_PID.State = 0);
   #FP_DIM.AutoTune_Undo := NOT #FP_PARM_TIA.AutoTune_SUT_Running AND NOT #FP_PARM_TIA.AutoTune_TIR_Running;
   #DummyBool := #FP_DIM.Auto AND #FP_DIM.Manual AND #FP_DIM.Internal AND #FP_DIM.Cascade AND #FP_SHOW.PB_LastSP AND #FP_DIM.AutoTune_Start_TIR AND #FP_DIM.AutoTune_Ack AND #FP_DIM.AutoTune_Undo;
END_REGION

REGION Network 10: Save Current State
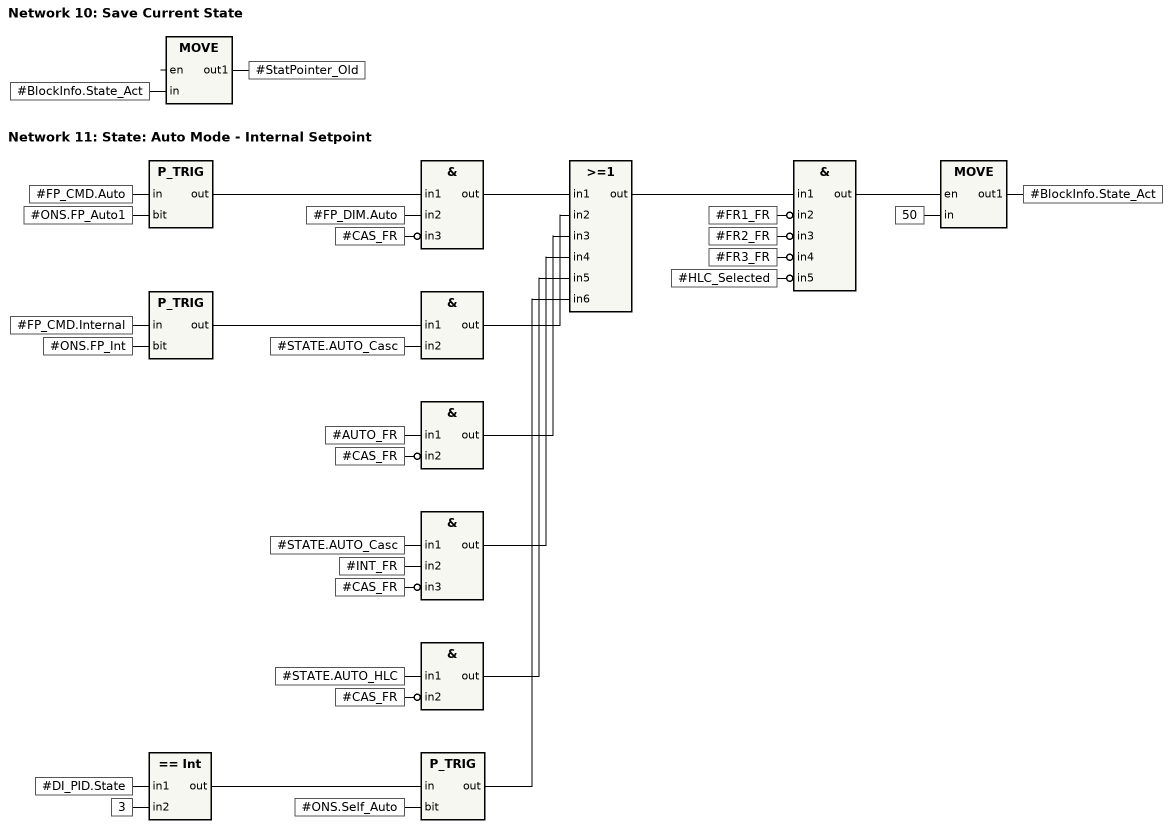
   #StatPointer_Old := #BlockInfo.State_Act;
END_REGION

REGION Network 11: State: Auto Mode - Internal Setpoint
   #_w1 := #FP_CMD.Auto AND NOT #ONS.FP_Auto1;   // rising edge
   #ONS.FP_Auto1 := #FP_CMD.Auto;
   #_w2 := #FP_CMD.Internal AND NOT #ONS.FP_Int;   // rising edge
   #ONS.FP_Int := #FP_CMD.Internal;
   #_w3 := #DI_PID.State = 3;
   #_w4 := #_w3 AND NOT #ONS.Self_Auto;   // rising edge
   #ONS.Self_Auto := #_w3;
   IF ((#_w1 AND #FP_DIM.Auto AND NOT #CAS_FR) OR (#_w2 AND #STATE.AUTO_Casc) OR (#AUTO_FR AND NOT #CAS_FR) OR (#STATE.AUTO_Casc AND #INT_FR AND NOT #CAS_FR) OR (#STATE.AUTO_HLC AND NOT #CAS_FR) OR #_w4) AND NOT #FR1_FR AND NOT #FR2_FR AND NOT #FR3_FR AND NOT #HLC_Selected THEN
       #BlockInfo.State_Act := 50;
   END_IF;
END_REGION

REGION Network 12: State: Auto Mode - Cascade Setpoint
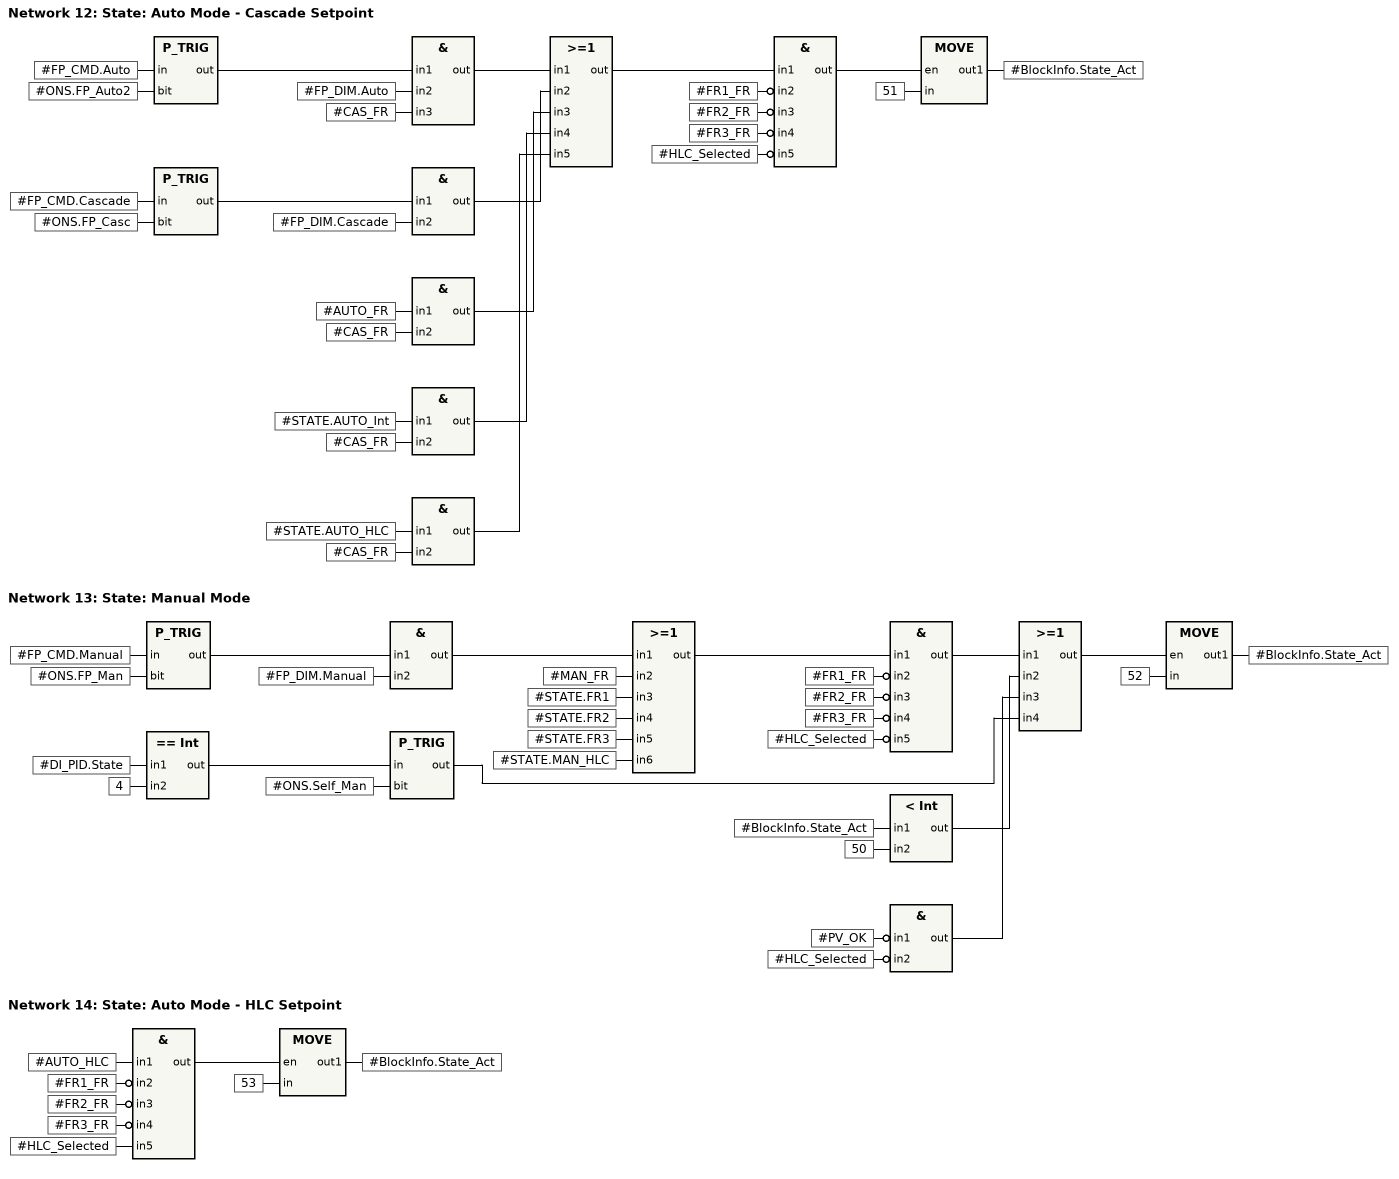
   #_w1 := #FP_CMD.Auto AND NOT #ONS.FP_Auto2;   // rising edge
   #ONS.FP_Auto2 := #FP_CMD.Auto;
   #_w2 := #FP_CMD.Cascade AND NOT #ONS.FP_Casc;   // rising edge
   #ONS.FP_Casc := #FP_CMD.Cascade;
   IF ((#_w1 AND #FP_DIM.Auto AND #CAS_FR) OR (#_w2 AND #FP_DIM.Cascade) OR (#AUTO_FR AND #CAS_FR) OR (#STATE.AUTO_Int AND #CAS_FR) OR (#STATE.AUTO_HLC AND #CAS_FR)) AND NOT #FR1_FR AND NOT #FR2_FR AND NOT #FR3_FR AND NOT #HLC_Selected THEN
       #BlockInfo.State_Act := 51;
   END_IF;
END_REGION

REGION Network 13: State: Manual Mode
   #_w1 := #FP_CMD.Manual AND NOT #ONS.FP_Man;   // rising edge
   #ONS.FP_Man := #FP_CMD.Manual;
   #_w2 := #DI_PID.State = 4;
   #_w3 := #_w2 AND NOT #ONS.Self_Man;   // rising edge
   #ONS.Self_Man := #_w2;
   IF (((#_w1 AND #FP_DIM.Manual) OR #MAN_FR OR #STATE.FR1 OR #STATE.FR2 OR #STATE.FR3 OR #STATE.MAN_HLC) AND NOT #FR1_FR AND NOT #FR2_FR AND NOT #FR3_FR AND NOT #HLC_Selected) OR (#BlockInfo.State_Act < 50) OR (NOT #PV_OK AND NOT #HLC_Selected) OR #_w3 THEN
       #BlockInfo.State_Act := 52;
   END_IF;
END_REGION

REGION Network 14: State: Auto Mode - HLC Setpoint
   IF #AUTO_HLC AND NOT #FR1_FR AND NOT #FR2_FR AND NOT #FR3_FR AND #HLC_Selected THEN
       #BlockInfo.State_Act := 53;
   END_IF;
END_REGION

REGION Network 15: State: Manual Mode - HLC
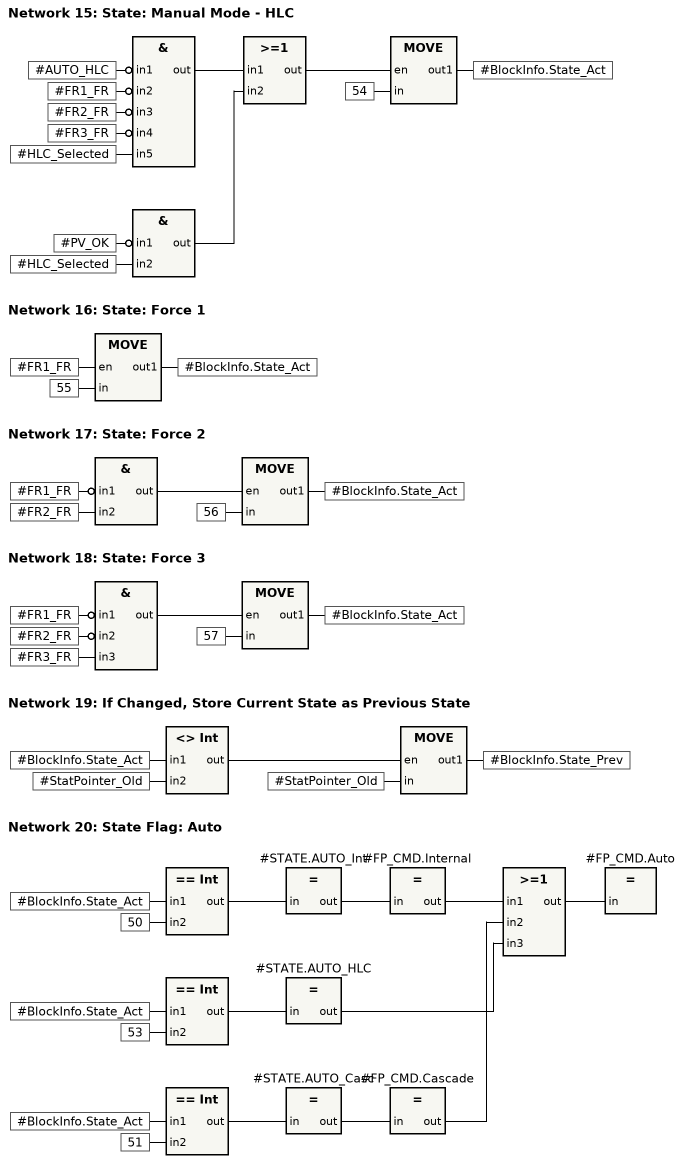
   IF (NOT #AUTO_HLC AND NOT #FR1_FR AND NOT #FR2_FR AND NOT #FR3_FR AND #HLC_Selected) OR (NOT #PV_OK AND #HLC_Selected) THEN
       #BlockInfo.State_Act := 54;
   END_IF;
END_REGION

REGION Network 16: State: Force 1
   IF #FR1_FR THEN #BlockInfo.State_Act := 55; END_IF;
END_REGION

REGION Network 17: State: Force 2
   IF NOT #FR1_FR AND #FR2_FR THEN #BlockInfo.State_Act := 56; END_IF;
END_REGION

REGION Network 18: State: Force 3
   IF NOT #FR1_FR AND NOT #FR2_FR AND #FR3_FR THEN #BlockInfo.State_Act := 57; END_IF;
END_REGION

REGION Network 19: If Changed, Store Current State as Previous State
   IF #BlockInfo.State_Act <> #StatPointer_Old THEN #BlockInfo.State_Prev := #StatPointer_Old; END_IF;
END_REGION

REGION Network 20: State Flag: Auto
   // >>>>> SET STATE FLAGS <<<<<
   #STATE.AUTO_Int := #BlockInfo.State_Act = 50;
   #FP_CMD.Internal := #STATE.AUTO_Int;
   #STATE.AUTO_Casc := #BlockInfo.State_Act = 51;
   #FP_CMD.Cascade := #STATE.AUTO_Casc;
   #STATE.AUTO_HLC := #BlockInfo.State_Act = 53;
   #FP_CMD.Auto := #STATE.AUTO_Int OR #STATE.AUTO_Casc OR #STATE.AUTO_HLC;
END_REGION

REGION Network 21: State Flag: Manual
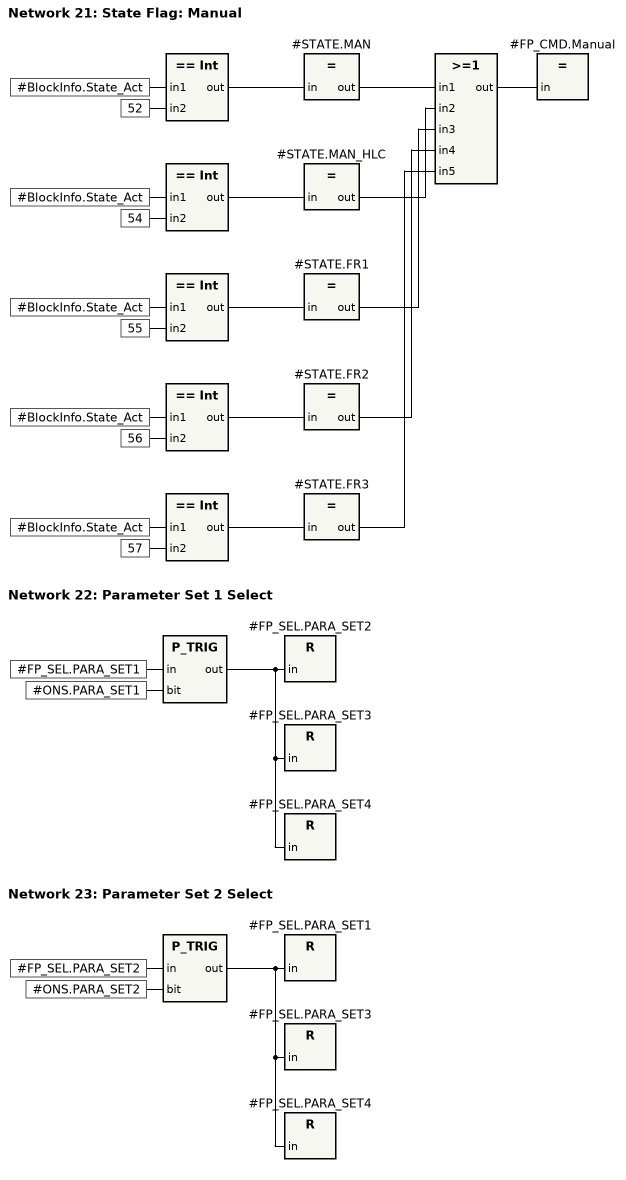
   #STATE.MAN := #BlockInfo.State_Act = 52;
   #STATE.MAN_HLC := #BlockInfo.State_Act = 54;
   #STATE.FR1 := #BlockInfo.State_Act = 55;
   #STATE.FR2 := #BlockInfo.State_Act = 56;
   #STATE.FR3 := #BlockInfo.State_Act = 57;
   #FP_CMD.Manual := #STATE.MAN OR #STATE.MAN_HLC OR #STATE.FR1 OR #STATE.FR2 OR #STATE.FR3;
END_REGION

REGION Network 22: Parameter Set 1 Select
   // >>>>> PARAMETER SELECT <<<<<
   #_w1 := #FP_SEL.PARA_SET1 AND NOT #ONS.PARA_SET1;   // rising edge
   #ONS.PARA_SET1 := #FP_SEL.PARA_SET1;
   IF #_w1 THEN
       #FP_SEL.PARA_SET2 := FALSE;
       #FP_SEL.PARA_SET3 := FALSE;
       #FP_SEL.PARA_SET4 := FALSE;
   END_IF;
END_REGION

REGION Network 23: Parameter Set 2 Select
   #_w1 := #FP_SEL.PARA_SET2 AND NOT #ONS.PARA_SET2;   // rising edge
   #ONS.PARA_SET2 := #FP_SEL.PARA_SET2;
   IF #_w1 THEN
       #FP_SEL.PARA_SET1 := FALSE;
       #FP_SEL.PARA_SET3 := FALSE;
       #FP_SEL.PARA_SET4 := FALSE;
   END_IF;
END_REGION

REGION Network 24: Parameter Set 3 Select
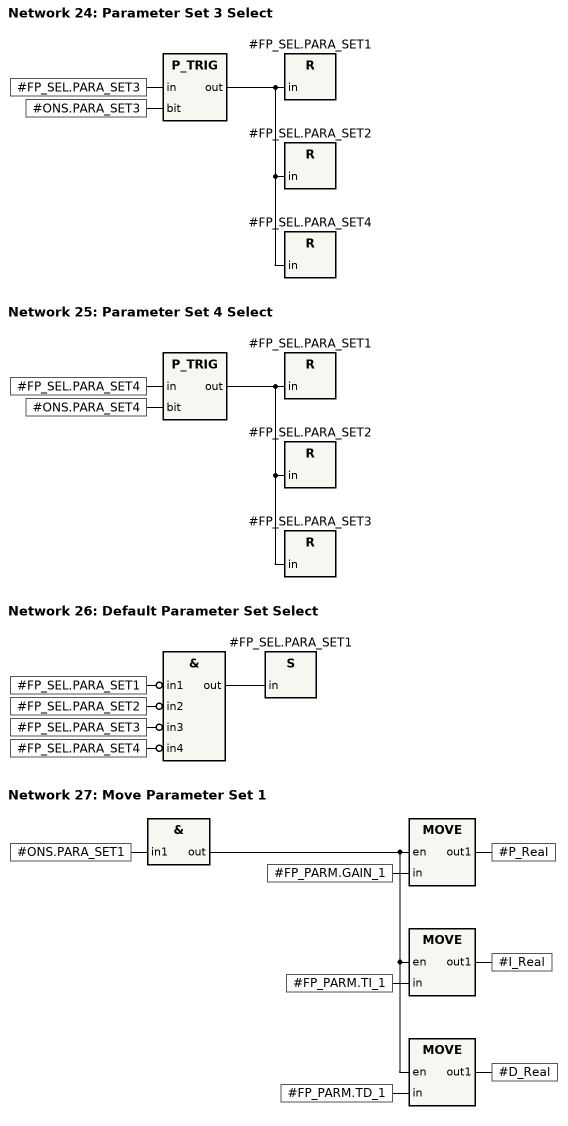
   #_w1 := #FP_SEL.PARA_SET3 AND NOT #ONS.PARA_SET3;   // rising edge
   #ONS.PARA_SET3 := #FP_SEL.PARA_SET3;
   IF #_w1 THEN
       #FP_SEL.PARA_SET1 := FALSE;
       #FP_SEL.PARA_SET2 := FALSE;
       #FP_SEL.PARA_SET4 := FALSE;
   END_IF;
END_REGION

REGION Network 25: Parameter Set 4 Select
   #_w1 := #FP_SEL.PARA_SET4 AND NOT #ONS.PARA_SET4;   // rising edge
   #ONS.PARA_SET4 := #FP_SEL.PARA_SET4;
   IF #_w1 THEN
       #FP_SEL.PARA_SET1 := FALSE;
       #FP_SEL.PARA_SET2 := FALSE;
       #FP_SEL.PARA_SET3 := FALSE;
   END_IF;
END_REGION

REGION Network 26: Default Parameter Set Select
   IF NOT #FP_SEL.PARA_SET1 AND NOT #FP_SEL.PARA_SET2 AND NOT #FP_SEL.PARA_SET3 AND NOT #FP_SEL.PARA_SET4 THEN
       #FP_SEL.PARA_SET1 := TRUE;
   END_IF;
END_REGION

REGION Network 27: Move Parameter Set 1
   IF #ONS.PARA_SET1 THEN
       #P_Real := #FP_PARM.GAIN_1;
       #I_Real := #FP_PARM.TI_1;
       #D_Real := #FP_PARM.TD_1;
   END_IF;
END_REGION

REGION Network 28: Move Parameter Set 2
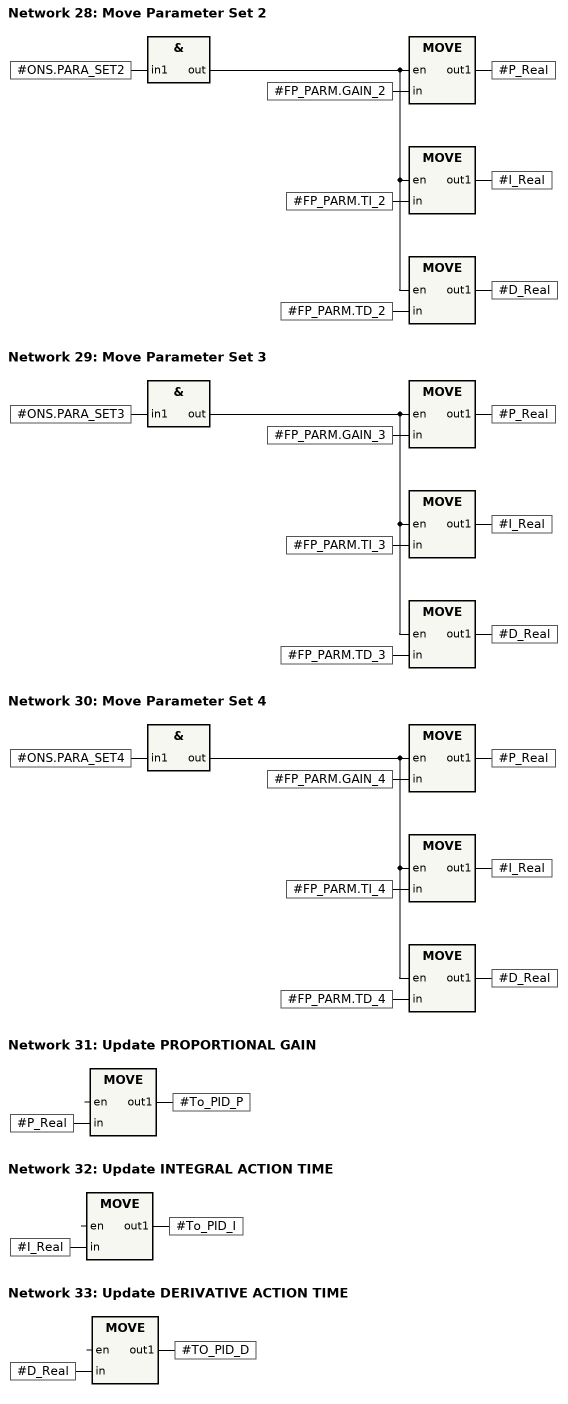
   IF #ONS.PARA_SET2 THEN
       #P_Real := #FP_PARM.GAIN_2;
       #I_Real := #FP_PARM.TI_2;
       #D_Real := #FP_PARM.TD_2;
   END_IF;
END_REGION

REGION Network 29: Move Parameter Set 3
   IF #ONS.PARA_SET3 THEN
       #P_Real := #FP_PARM.GAIN_3;
       #I_Real := #FP_PARM.TI_3;
       #D_Real := #FP_PARM.TD_3;
   END_IF;
END_REGION

REGION Network 30: Move Parameter Set 4
   IF #ONS.PARA_SET4 THEN
       #P_Real := #FP_PARM.GAIN_4;
       #I_Real := #FP_PARM.TI_4;
       #D_Real := #FP_PARM.TD_4;
   END_IF;
END_REGION

REGION Network 31: Update PROPORTIONAL GAIN
   #To_PID_P := #P_Real;
END_REGION

REGION Network 32: Update INTEGRAL ACTION TIME
   #To_PID_I := #I_Real;
END_REGION

REGION Network 33: Update DERIVATIVE ACTION TIME
   #TO_PID_D := #D_Real;
END_REGION

REGION Network 34: Feed Forward Calculation
   // >>>>> FEED FORWARD <<<<<
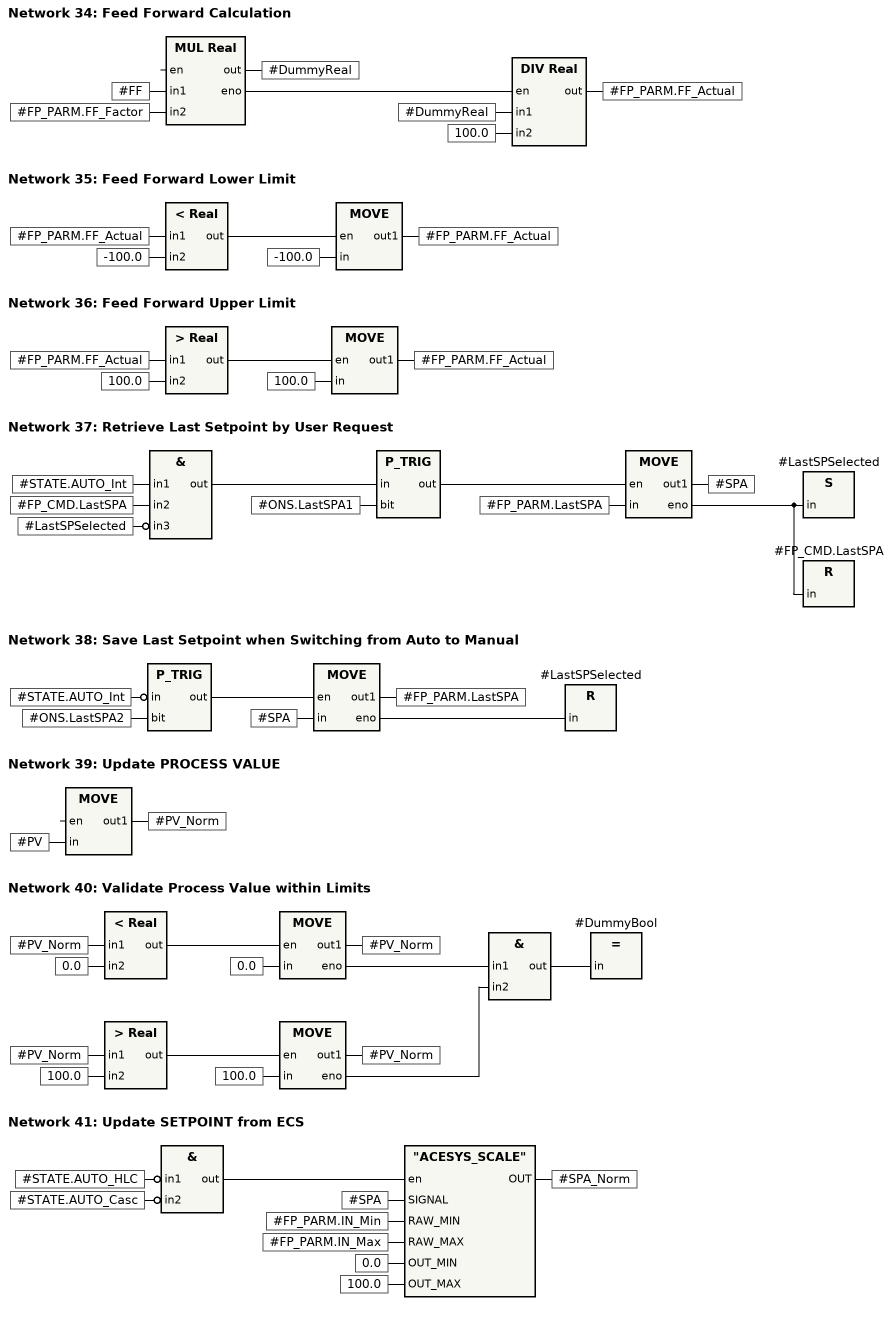
   // ENO of a box is taken as its EN; it also drops when the box reports an error
   #DummyReal := #FF * #FP_PARM.FF_Factor;
   #FP_PARM.FF_Actual := #DummyReal / 100.0;
END_REGION

REGION Network 35: Feed Forward Lower Limit
   IF #FP_PARM.FF_Actual < (-100.0) THEN #FP_PARM.FF_Actual := -100.0; END_IF;
END_REGION

REGION Network 36: Feed Forward Upper Limit
   IF #FP_PARM.FF_Actual > 100.0 THEN #FP_PARM.FF_Actual := 100.0; END_IF;
END_REGION

REGION Network 37: Retrieve Last Setpoint by User Request
   // >>>>> LAST SP <<<<<
   // ENO of a box is taken as its EN; it also drops when the box reports an error
   #_w1 := #STATE.AUTO_Int AND #FP_CMD.LastSPA AND NOT #LastSPSelected;
   #_w2 := #_w1 AND NOT #ONS.LastSPA1;   // rising edge
   #ONS.LastSPA1 := #_w1;
   IF #_w2 THEN
       #SPA := #FP_PARM.LastSPA;
       #LastSPSelected := TRUE;
       #FP_CMD.LastSPA := FALSE;
   END_IF;
END_REGION

REGION Network 38: Save Last Setpoint when Switching from Auto to Manual
   // ENO of a box is taken as its EN; it also drops when the box reports an error
   #_w1 := NOT #STATE.AUTO_Int AND NOT #ONS.LastSPA2;   // rising edge
   #ONS.LastSPA2 := NOT #STATE.AUTO_Int;
   IF #_w1 THEN
       #FP_PARM.LastSPA := #SPA;
       #LastSPSelected := FALSE;
   END_IF;
END_REGION

REGION Network 39: Update PROCESS VALUE
   // >>>>> PROCESS VALUE <<<<<
   #PV_Norm := #PV;
END_REGION

REGION Network 40: Validate Process Value within Limits
   // ENO of a box is taken as its EN; it also drops when the box reports an error
   #_w1 := #PV_Norm < 0.0;
   IF #_w1 THEN #PV_Norm := 0.0; END_IF;
   #_w2 := #PV_Norm > 100.0;
   IF #_w2 THEN #PV_Norm := 100.0; END_IF;
   #DummyBool := #_w1 AND #_w2;
END_REGION

REGION Network 41: Update SETPOINT from ECS
   // >>>>> SPA Selection <<<<<
   IF NOT #STATE.AUTO_HLC AND NOT #STATE.AUTO_Casc THEN
       "ACESYS_SCALE"(SIGNAL := #SPA,
                      RAW_MIN := #FP_PARM.IN_Min,
                      RAW_MAX := #FP_PARM.IN_Max,
                      OUT_MIN := 0.0,
                      OUT_MAX := 100.0,
                      OUT => #SPA_Norm);
   END_IF;
END_REGION

REGION Network 42: Update SETPOINT from Cascade
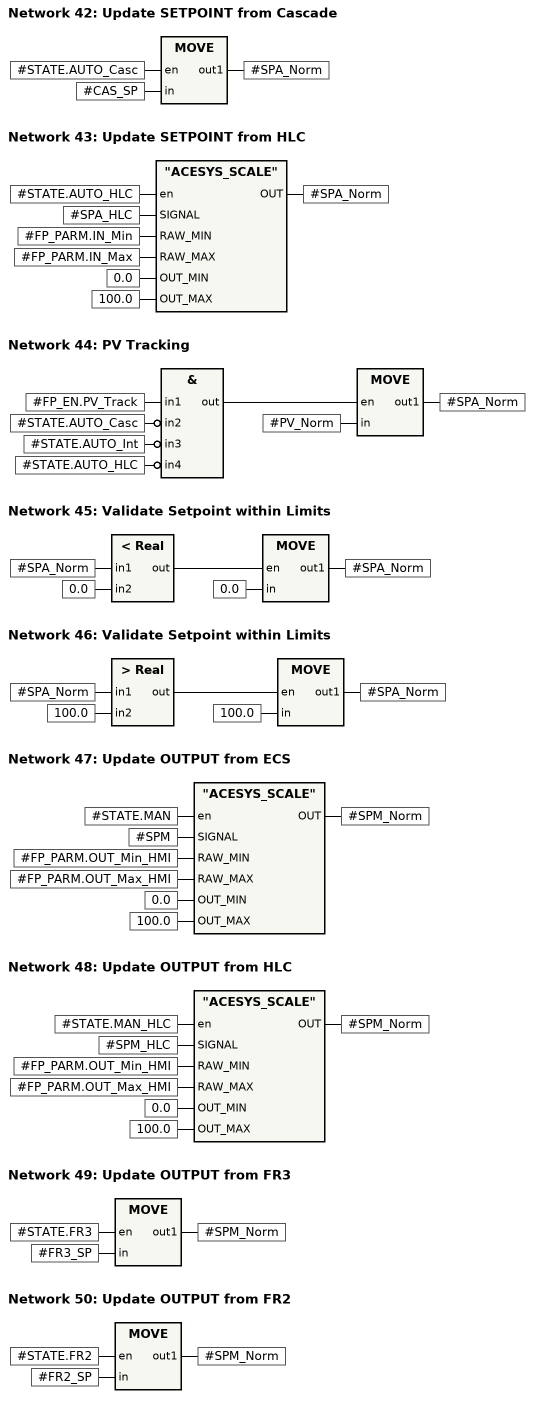
   IF #STATE.AUTO_Casc THEN #SPA_Norm := #CAS_SP; END_IF;
END_REGION

REGION Network 43: Update SETPOINT from HLC
   IF #STATE.AUTO_HLC THEN
       "ACESYS_SCALE"(SIGNAL := #SPA_HLC,
                      RAW_MIN := #FP_PARM.IN_Min,
                      RAW_MAX := #FP_PARM.IN_Max,
                      OUT_MIN := 0.0,
                      OUT_MAX := 100.0,
                      OUT => #SPA_Norm);
   END_IF;
END_REGION

REGION Network 44: PV Tracking
   IF #FP_EN.PV_Track AND NOT #STATE.AUTO_Casc AND NOT #STATE.AUTO_Int AND NOT #STATE.AUTO_HLC THEN
       #SPA_Norm := #PV_Norm;
   END_IF;
END_REGION

REGION Network 45: Validate Setpoint within Limits
   IF #SPA_Norm < 0.0 THEN #SPA_Norm := 0.0; END_IF;
END_REGION

REGION Network 46: Validate Setpoint within Limits
   IF #SPA_Norm > 100.0 THEN #SPA_Norm := 100.0; END_IF;
END_REGION

REGION Network 47: Update OUTPUT from ECS
   // >>>>> SPM SELECTION <<<<<
   IF #STATE.MAN THEN
       "ACESYS_SCALE"(SIGNAL := #SPM,
                      RAW_MIN := #FP_PARM.OUT_Min_HMI,
                      RAW_MAX := #FP_PARM.OUT_Max_HMI,
                      OUT_MIN := 0.0,
                      OUT_MAX := 100.0,
                      OUT => #SPM_Norm);
   END_IF;
END_REGION

REGION Network 48: Update OUTPUT from HLC
   // Build 004 - 09. Marts 2016 (FKP) : New network
   IF #STATE.MAN_HLC THEN
       "ACESYS_SCALE"(SIGNAL := #SPM_HLC,
                      RAW_MIN := #FP_PARM.OUT_Min_HMI,
                      RAW_MAX := #FP_PARM.OUT_Max_HMI,
                      OUT_MIN := 0.0,
                      OUT_MAX := 100.0,
                      OUT => #SPM_Norm);
   END_IF;
END_REGION

REGION Network 49: Update OUTPUT from FR3
   IF #STATE.FR3 THEN #SPM_Norm := #FR3_SP; END_IF;
END_REGION

REGION Network 50: Update OUTPUT from FR2
   IF #STATE.FR2 THEN #SPM_Norm := #FR2_SP; END_IF;
END_REGION

REGION Network 51: Update OUTPUT from FR1
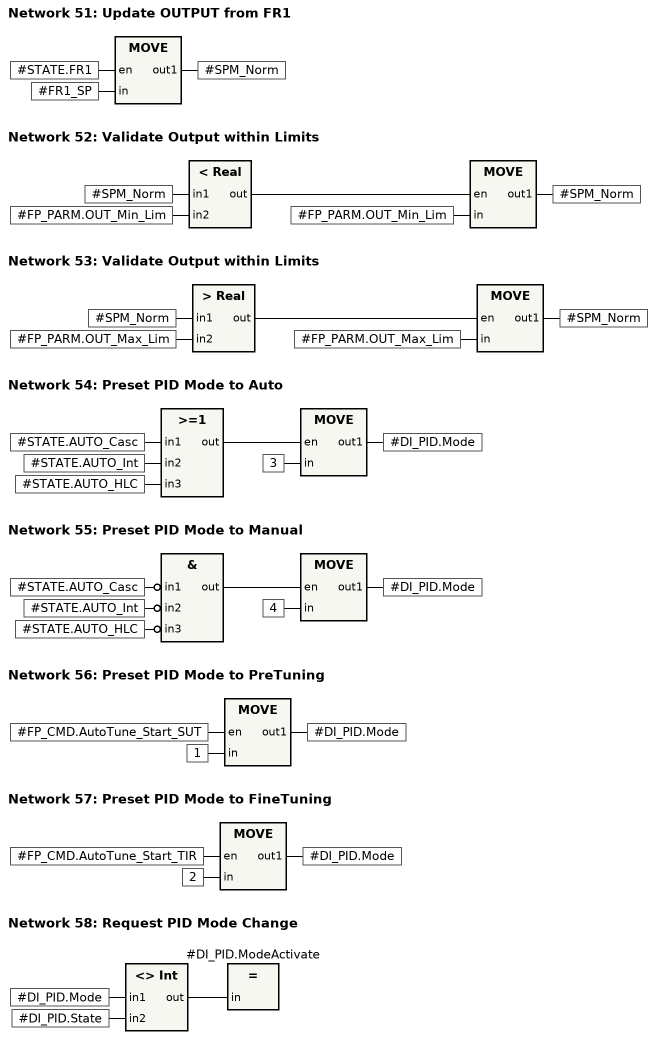
   IF #STATE.FR1 THEN #SPM_Norm := #FR1_SP; END_IF;
END_REGION

REGION Network 52: Validate Output within Limits
   // Build 002 - 4.Oct.2015 : Move var changed from #FP_PARM.OUT_Min_HMI to
   //                           #FP_PARM.OUT_Min_Lim
   IF #SPM_Norm < #FP_PARM.OUT_Min_Lim THEN #SPM_Norm := #FP_PARM.OUT_Min_Lim; END_IF;
END_REGION

REGION Network 53: Validate Output within Limits
   // Build 002 - 4.Oct.2015 : Move var changed from #FP_PARM.OUT_Max_HMI to
   //                         #FP_PARM.OUT_Max_Lim
   IF #SPM_Norm > #FP_PARM.OUT_Max_Lim THEN #SPM_Norm := #FP_PARM.OUT_Max_Lim; END_IF;
END_REGION

REGION Network 54: Preset PID Mode to Auto
   IF #STATE.AUTO_Casc OR #STATE.AUTO_Int OR #STATE.AUTO_HLC THEN #DI_PID.Mode := 3; END_IF;
END_REGION

REGION Network 55: Preset PID Mode to Manual
   // >>>>> Set PID to Manual Mode <<<<<
   IF NOT #STATE.AUTO_Casc AND NOT #STATE.AUTO_Int AND NOT #STATE.AUTO_HLC THEN #DI_PID.Mode := 4; END_IF;
END_REGION

REGION Network 56: Preset PID Mode to PreTuning
   IF #FP_CMD.AutoTune_Start_SUT THEN #DI_PID.Mode := 1; END_IF;
END_REGION

REGION Network 57: Preset PID Mode to FineTuning
   IF #FP_CMD.AutoTune_Start_TIR THEN #DI_PID.Mode := 2; END_IF;
END_REGION

REGION Network 58: Request PID Mode Change
   #DI_PID.ModeActivate := #DI_PID.Mode <> #DI_PID.State;
END_REGION

REGION Network 59: PID Parameterization
   // >>>>> MOVE PARAMETERS TO PID <<<<<
   // Build 003 - 26. Oct 2021 (BOBO-IN) : PID Configurable Cycle time added newly
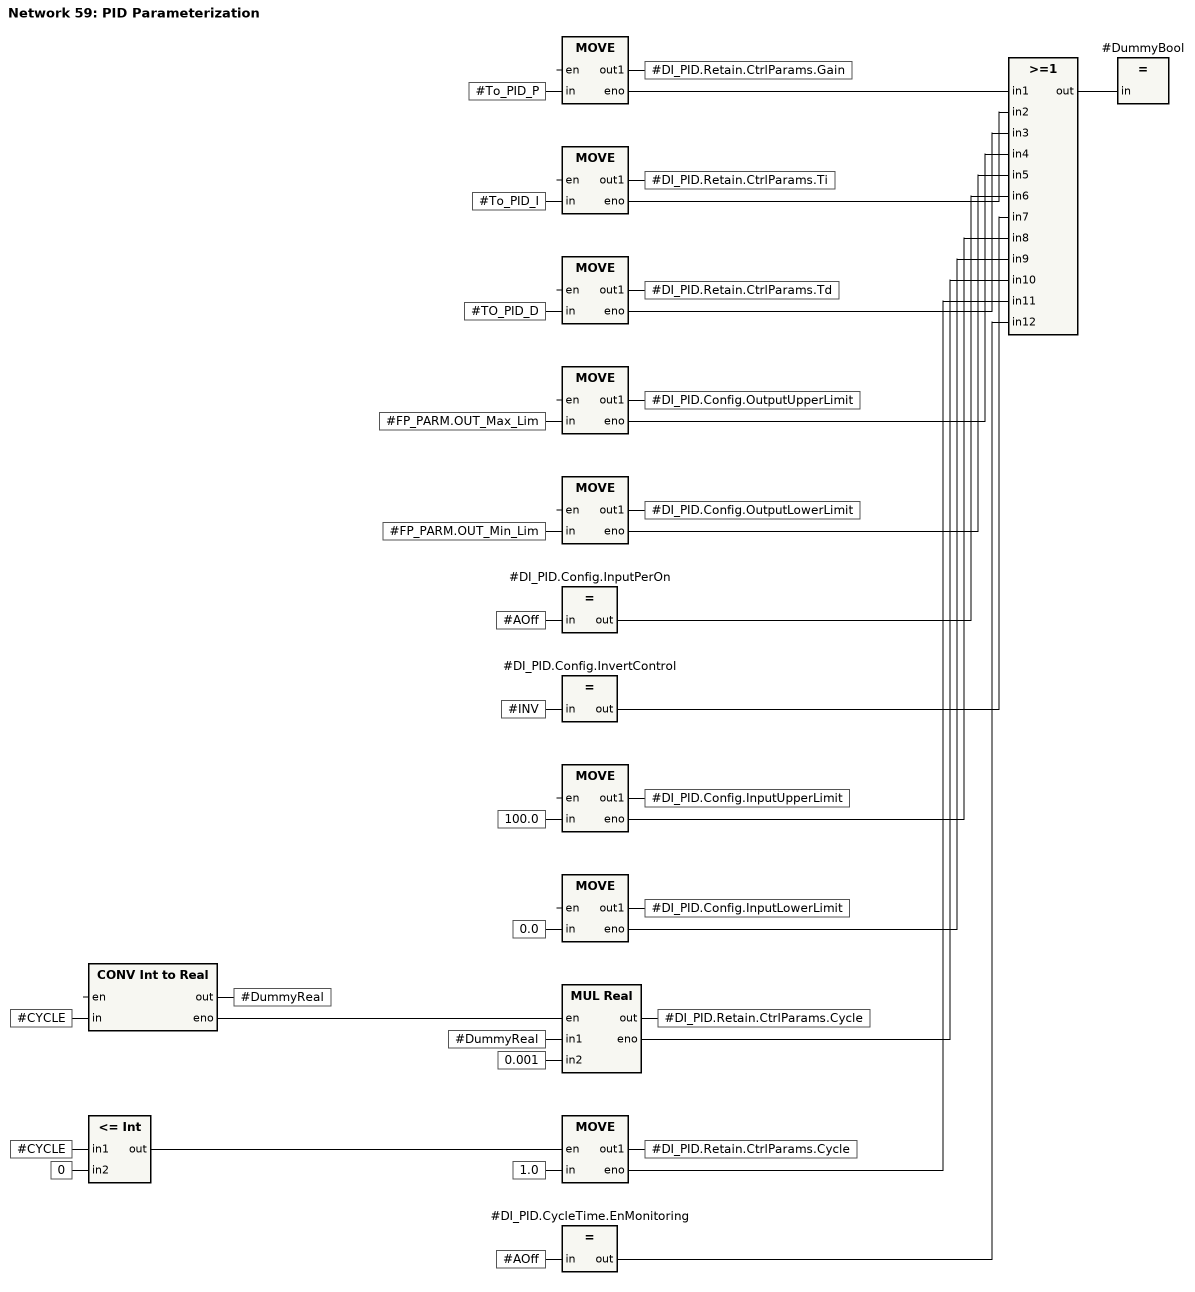
   #DI_PID.Retain.CtrlParams.Gain := #To_PID_P;
   #DI_PID.Retain.CtrlParams.Ti := #To_PID_I;
   #DI_PID.Retain.CtrlParams.Td := #TO_PID_D;
   #DI_PID.Config.OutputUpperLimit := #FP_PARM.OUT_Max_Lim;
   #DI_PID.Config.OutputLowerLimit := #FP_PARM.OUT_Min_Lim;
   #DI_PID.Config.InputPerOn := #AOff;
   #DI_PID.Config.InvertControl := #INV;
   #DI_PID.Config.InputUpperLimit := 100.0;
   #DI_PID.Config.InputLowerLimit := 0.0;
   #DummyReal := INT_TO_REAL(#CYCLE);
   #DI_PID.Retain.CtrlParams.Cycle := #DummyReal * 0.001;
   #_w1 := #CYCLE <= 0;
   IF #_w1 THEN #DI_PID.Retain.CtrlParams.Cycle := 1.0; END_IF;
   #DI_PID.CycleTime.EnMonitoring := #AOff;
   #DummyBool := TRUE OR TRUE OR TRUE OR TRUE OR TRUE OR #AOff OR #INV OR TRUE OR TRUE OR TRUE OR #_w1 OR #AOff;
END_REGION

REGION Network 60: Deadband Logic
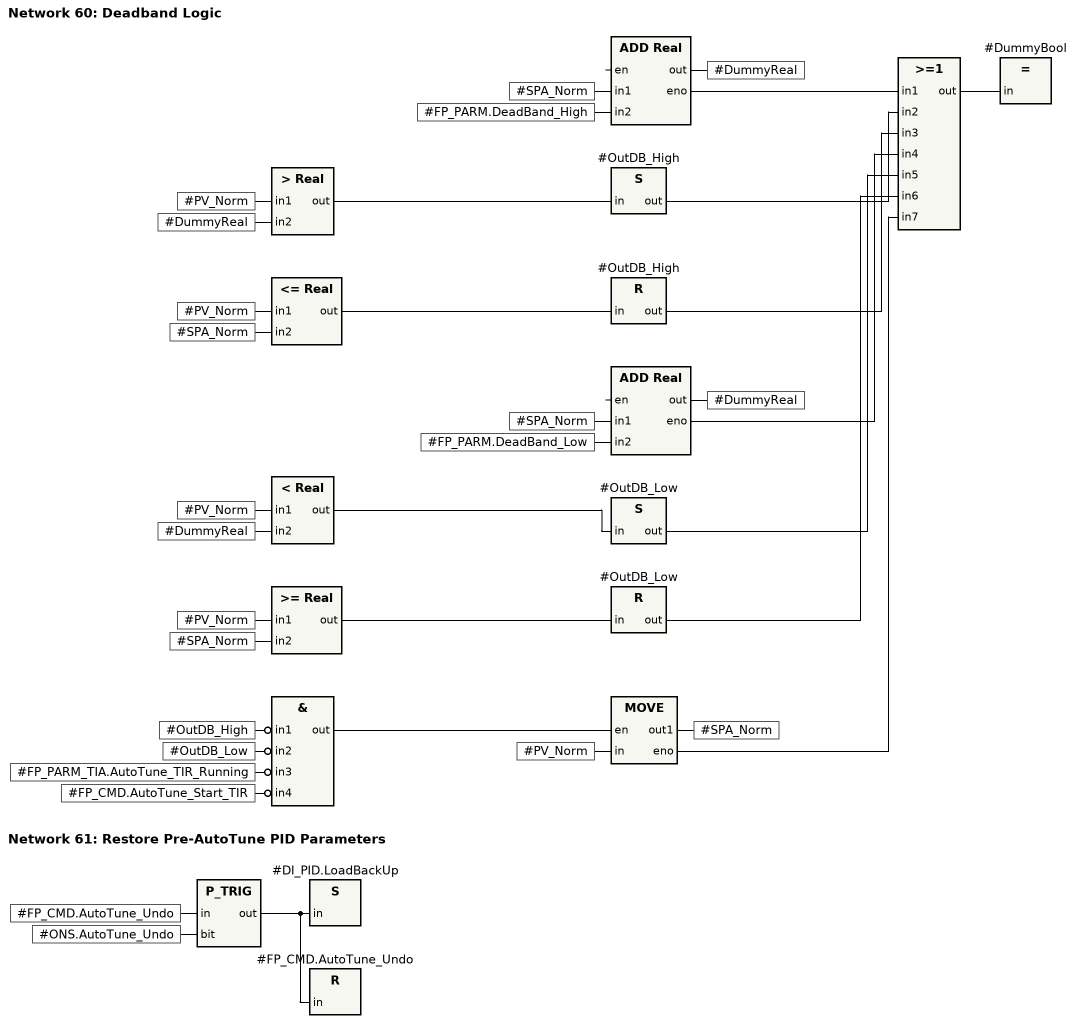
   #DummyReal := #SPA_Norm + #FP_PARM.DeadBand_High;
   #_w1 := #PV_Norm > #DummyReal;
   IF #_w1 THEN #OutDB_High := TRUE; END_IF;
   #_w2 := #PV_Norm <= #SPA_Norm;
   IF #_w2 THEN #OutDB_High := FALSE; END_IF;
   #DummyReal := #SPA_Norm + #FP_PARM.DeadBand_Low;
   #_w3 := #PV_Norm < #DummyReal;
   IF #_w3 THEN #OutDB_Low := TRUE; END_IF;
   #_w4 := #PV_Norm >= #SPA_Norm;
   IF #_w4 THEN #OutDB_Low := FALSE; END_IF;
   #_w5 := NOT #OutDB_High AND NOT #OutDB_Low AND NOT #FP_PARM_TIA.AutoTune_TIR_Running AND NOT #FP_CMD.AutoTune_Start_TIR;
   IF #_w5 THEN #SPA_Norm := #PV_Norm; END_IF;
   #DummyBool := TRUE OR #_w1 OR #_w2 OR TRUE OR #_w3 OR #_w4 OR #_w5;
END_REGION

REGION Network 61: Restore Pre-AutoTune PID Parameters
   #_w1 := #FP_CMD.AutoTune_Undo AND NOT #ONS.AutoTune_Undo;   // rising edge
   #ONS.AutoTune_Undo := #FP_CMD.AutoTune_Undo;
   IF #_w1 THEN
       #DI_PID.LoadBackUp := TRUE;
       #FP_CMD.AutoTune_Undo := FALSE;
   END_IF;
END_REGION

REGION Network 62: PID
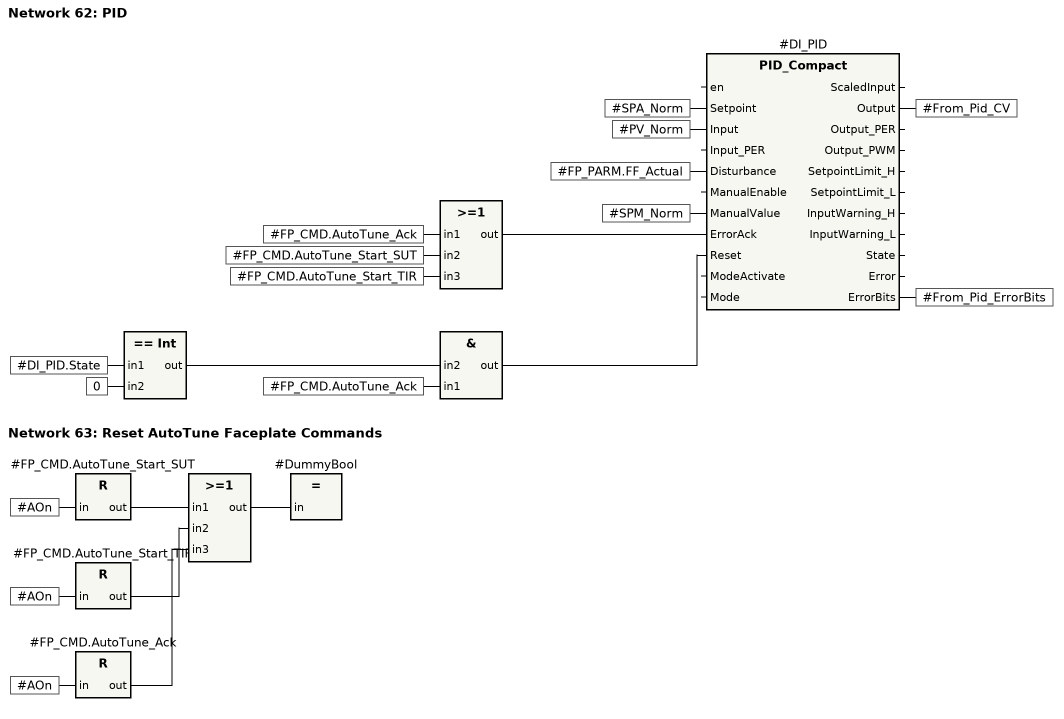
   #DI_PID(Setpoint := #SPA_Norm,   // PID_Compact
           Input := #PV_Norm,
           Disturbance := #FP_PARM.FF_Actual,
           ManualValue := #SPM_Norm,
           ErrorAck := #FP_CMD.AutoTune_Ack OR #FP_CMD.AutoTune_Start_SUT OR #FP_CMD.AutoTune_Start_TIR,
           Reset := (#DI_PID.State = 0) AND #FP_CMD.AutoTune_Ack,
           Output => #From_Pid_CV,
           ErrorBits => #From_Pid_ErrorBits);
END_REGION

REGION Network 63: Reset AutoTune Faceplate Commands
   IF #AOn THEN
       #FP_CMD.AutoTune_Start_SUT := FALSE;
       #FP_CMD.AutoTune_Start_TIR := FALSE;
       #FP_CMD.AutoTune_Ack := FALSE;
   END_IF;
   #DummyBool := #AOn OR #AOn OR #AOn;
END_REGION

REGION Network 64: Update Faceplate with AutoTune Results
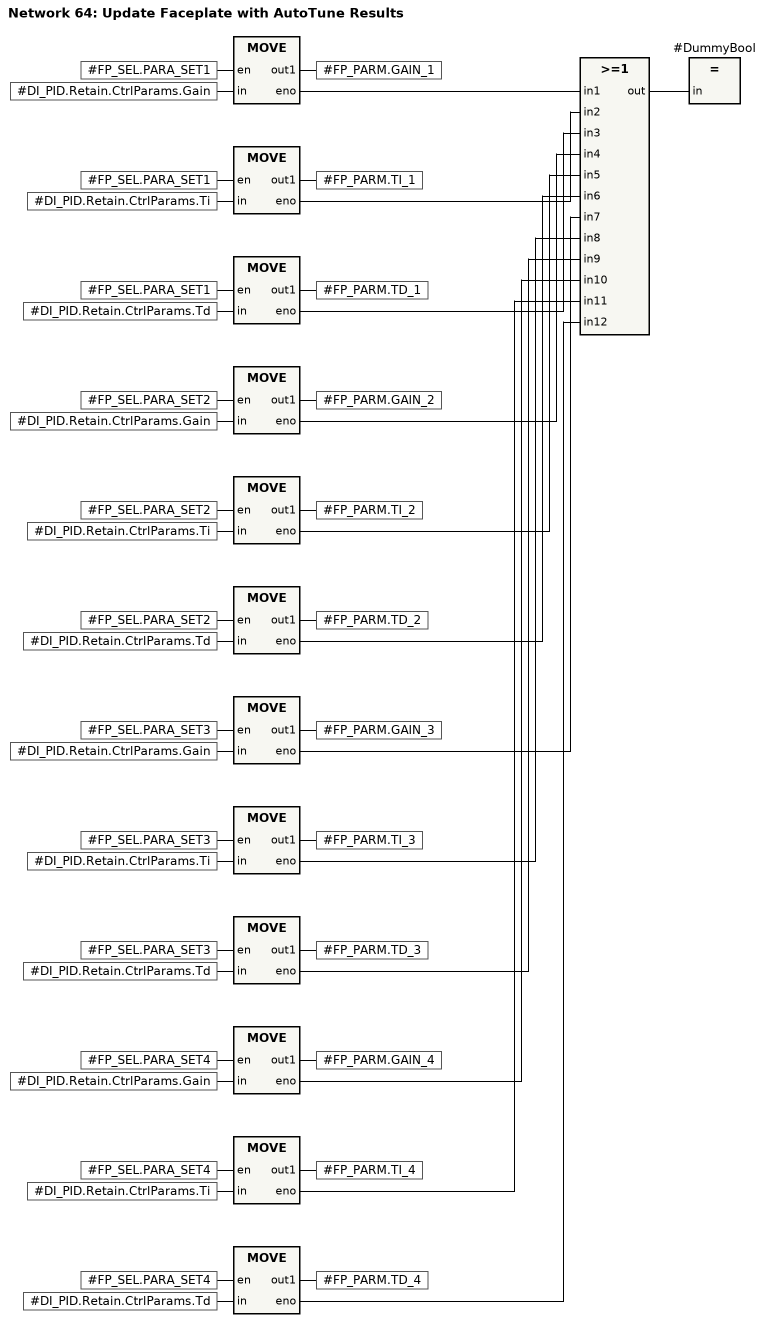
   IF #FP_SEL.PARA_SET1 THEN
       #FP_PARM.GAIN_1 := #DI_PID.Retain.CtrlParams.Gain;
       #FP_PARM.TI_1 := #DI_PID.Retain.CtrlParams.Ti;
       #FP_PARM.TD_1 := #DI_PID.Retain.CtrlParams.Td;
   END_IF;
   IF #FP_SEL.PARA_SET2 THEN
       #FP_PARM.GAIN_2 := #DI_PID.Retain.CtrlParams.Gain;
       #FP_PARM.TI_2 := #DI_PID.Retain.CtrlParams.Ti;
       #FP_PARM.TD_2 := #DI_PID.Retain.CtrlParams.Td;
   END_IF;
   IF #FP_SEL.PARA_SET3 THEN
       #FP_PARM.GAIN_3 := #DI_PID.Retain.CtrlParams.Gain;
       #FP_PARM.TI_3 := #DI_PID.Retain.CtrlParams.Ti;
       #FP_PARM.TD_3 := #DI_PID.Retain.CtrlParams.Td;
   END_IF;
   IF #FP_SEL.PARA_SET4 THEN
       #FP_PARM.GAIN_4 := #DI_PID.Retain.CtrlParams.Gain;
       #FP_PARM.TI_4 := #DI_PID.Retain.CtrlParams.Ti;
       #FP_PARM.TD_4 := #DI_PID.Retain.CtrlParams.Td;
   END_IF;
   #DummyBool := #FP_SEL.PARA_SET1 OR #FP_SEL.PARA_SET1 OR #FP_SEL.PARA_SET1 OR #FP_SEL.PARA_SET2 OR #FP_SEL.PARA_SET2 OR #FP_SEL.PARA_SET2 OR #FP_SEL.PARA_SET3 OR #FP_SEL.PARA_SET3 OR #FP_SEL.PARA_SET3 OR #FP_SEL.PARA_SET4 OR #FP_SEL.PARA_SET4 OR #FP_SEL.PARA_SET4;
END_REGION

REGION Network 65: Block Output: CV
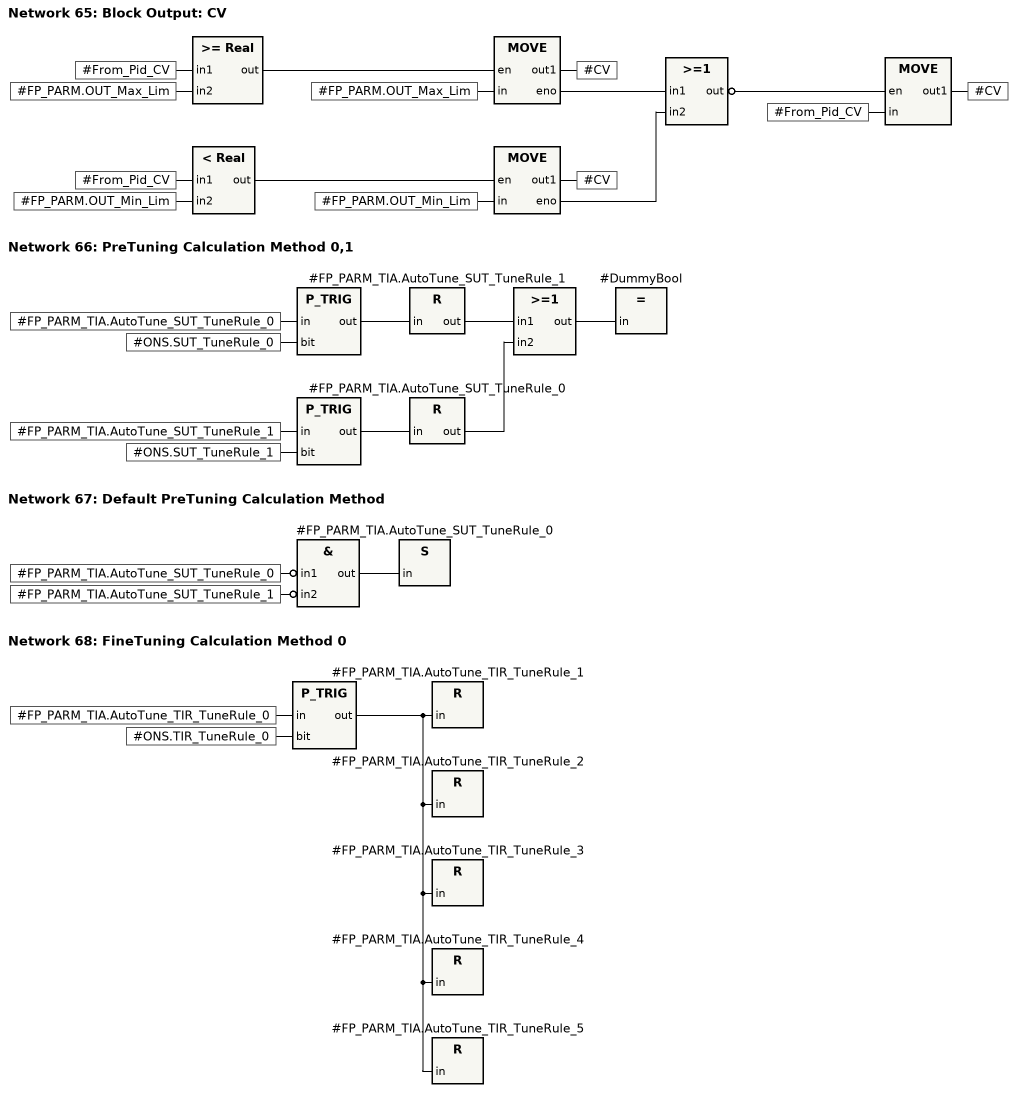
   // ENO of a box is taken as its EN; it also drops when the box reports an error
   #_w1 := #From_Pid_CV >= #FP_PARM.OUT_Max_Lim;
   IF #_w1 THEN #CV := #FP_PARM.OUT_Max_Lim; END_IF;
   #_w2 := #From_Pid_CV < #FP_PARM.OUT_Min_Lim;
   IF #_w2 THEN #CV := #FP_PARM.OUT_Min_Lim; END_IF;
   IF NOT (#_w1 OR #_w2) THEN #CV := #From_Pid_CV; END_IF;
END_REGION

REGION Network 66: PreTuning Calculation Method 0,1
   #_w1 := #FP_PARM_TIA.AutoTune_SUT_TuneRule_0 AND NOT #ONS.SUT_TuneRule_0;   // rising edge
   #ONS.SUT_TuneRule_0 := #FP_PARM_TIA.AutoTune_SUT_TuneRule_0;
   IF #_w1 THEN #FP_PARM_TIA.AutoTune_SUT_TuneRule_1 := FALSE; END_IF;
   #_w2 := #FP_PARM_TIA.AutoTune_SUT_TuneRule_1 AND NOT #ONS.SUT_TuneRule_1;   // rising edge
   #ONS.SUT_TuneRule_1 := #FP_PARM_TIA.AutoTune_SUT_TuneRule_1;
   IF #_w2 THEN #FP_PARM_TIA.AutoTune_SUT_TuneRule_0 := FALSE; END_IF;
   #DummyBool := #_w1 OR #_w2;
END_REGION

REGION Network 67: Default PreTuning Calculation Method
   IF NOT #FP_PARM_TIA.AutoTune_SUT_TuneRule_0 AND NOT #FP_PARM_TIA.AutoTune_SUT_TuneRule_1 THEN
       #FP_PARM_TIA.AutoTune_SUT_TuneRule_0 := TRUE;
   END_IF;
END_REGION

REGION Network 68: FineTuning Calculation Method 0
   #_w1 := #FP_PARM_TIA.AutoTune_TIR_TuneRule_0 AND NOT #ONS.TIR_TuneRule_0;   // rising edge
   #ONS.TIR_TuneRule_0 := #FP_PARM_TIA.AutoTune_TIR_TuneRule_0;
   IF #_w1 THEN
       #FP_PARM_TIA.AutoTune_TIR_TuneRule_1 := FALSE;
       #FP_PARM_TIA.AutoTune_TIR_TuneRule_2 := FALSE;
       #FP_PARM_TIA.AutoTune_TIR_TuneRule_3 := FALSE;
       #FP_PARM_TIA.AutoTune_TIR_TuneRule_4 := FALSE;
       #FP_PARM_TIA.AutoTune_TIR_TuneRule_5 := FALSE;
   END_IF;
END_REGION

REGION Network 69: FineTuning Calculation Method 1
